C01850=1115.478,64.441,-55.172,179.980,7.501,149.417
C01851=1115.474,64.655,-55.187,179.981,7.504,149.417
C01852=1115.470,64.869,-55.202,179.982,7.508,149.417
C01853=1115.464,65.119,-55.219,179.983,7.512,149.418
C01854=1115.460,65.367,-55.236,179.984,7.516,149.418
C01855=1115.454,65.617,-55.254,179.985,7.520,149.419
C01856=1115.450,65.867,-55.270,179.987,7.524,149.420
C01857=1115.445,66.116,-55.288,179.988,7.528,149.420
C01858=1115.440,66.366,-55.306,179.990,7.532,149.421
C01859=1115.436,66.615,-55.323,179.991,7.536,149.421
C01860=1115.430,66.864,-55.340,179.993,7.540,149.421
C01861=1115.425,67.114,-55.358,179.993,7.543,149.422
C01862=1115.421,67.363,-55.375,179.995,7.547,149.423
C01863=1115.415,67.612,-55.392,179.996,7.551,149.423
C01864=1115.410,67.861,-55.410,179.997,7.556,149.424
C01865=1115.406,68.111,-55.426,179.999,7.560,149.424
C01866=1115.401,68.360,-55.444,-179.999,7.563,149.425
C01867=1115.396,68.610,-55.462,-179.998,7.568,149.425
C01868=1115.391,68.859,-55.479,-179.997,7.572,149.426
C01869=1115.386,69.108,-55.496,-179.995,7.575,149.426
C01870=1115.381,69.358,-55.514,-179.994,7.580,149.427
C01871=1115.376,69.607,-55.532,-179.993,7.583,149.427
C01872=1115.372,69.856,-55.549,-179.991,7.587,149.428
C01873=1115.367,70.106,-55.566,-179.990,7.591,149.428
C01874=1115.362,70.355,-55.584,-179.989,7.595,149.429
C01875=1115.357,70.604,-55.602,-179.987,7.599,149.429
C01876=1115.352,70.854,-55.619,-179.986,7.603,149.430
C01877=1115.347,71.103,-55.637,-179.985,7.607,149.430
C01878=1115.342,71.353,-55.654,-179.983,7.611,149.431
C01879=1115.337,71.602,-55.672,-179.981,7.615,149.431
C01880=1115.333,71.851,-55.689,-179.980,7.619,149.432
C01881=1115.328,72.101,-55.707,-179.979,7.623,149.432
C01882=1115.323,72.350,-55.725,-179.977,7.627,149.433
C01883=1115.318,72.599,-55.743,-179.977,7.630,149.433
C01884=1115.313,72.849,-55.760,-179.975,7.634,149.434
C01885=1115.308,73.098,-55.778,-179.973,7.638,149.434
C01886=1115.304,73.347,-55.795,-179.972,7.643,149.435
C01887=1115.299,73.597,-55.813,-179.971,7.646,149.435
C01888=1115.294,73.846,-55.831,-179.969,7.650,149.436
C01889=1115.289,74.095,-55.848,-179.968,7.654,149.436
C01890=1115.284,74.344,-55.866,-179.967,7.659,149.437
C01891=1115.279,74.594,-55.884,-179.965,7.662,149.437
C01892=1115.274,74.843,-55.902,-179.963,7.666,149.437
C01893=1115.270,75.092,-55.919,-179.962,7.670,149.438
C01894=1115.265,75.341,-55.937,-179.961,7.675,149.439
C01895=1115.259,75.591,-55.954,-179.959,7.678,149.439
C01896=1115.254,75.840,-55.972,-179.958,7.682,149.439
C01897=1115.250,76.089,-55.990,-179.956,7.686,149.440
C01898=1115.245,76.338,-56.008,-179.955,7.690,149.440
C01899=1115.240,76.588,-56.026,-179.954,7.694,149.441
C01900=1115.235,76.837,-56.044,-179.952,7.698,149.441
C01901=1115.231,77.052,-56.060,-179.951,7.701,149.442
C01902=1115.227,77.266,-56.075,-179.951,7.704,149.442
C01903=1115.222,77.480,-56.090,-179.950,7.707,149.443
C01904=1115.219,77.694,-56.106,-179.949,7.710,149.443
C01905=1115.214,77.908,-56.121,-179.948,7.714,149.444
C01906=1115.210,78.123,-56.136,-179.947,7.717,149.444
C01907=1115.206,78.337,-56.152,-179.946,7.720,149.445
C01908=1115.201,78.551,-56.167,-179.946,7.723,149.445
C01909=1115.196,78.800,-56.185,-179.944,7.728,149.446
C01910=1115.192,79.049,-56.203,-179.943,7.731,149.446
C01911=1115.187,79.298,-56.221,-179.942,7.735,149.447
C01912=1115.182,79.548,-56.239,-179.941,7.738,149.447
C01913=1115.177,79.798,-56.257,-179.940,7.742,149.448
C01914=1115.173,80.047,-56.275,-179.939,7.745,149.448
C01915=1115.168,80.296,-56.293,-179.938,7.750,149.449
C01916=1115.163,80.545,-56.311,-179.937,7.753,149.450
C01917=1115.158,80.794,-56.329,-179.936,7.757,149.450
C01918=1115.153,81.043,-56.347,-179.935,7.760,149.451
C01919=1115.149,81.293,-56.366,-179.934,7.764,149.451
C01920=1115.144,81.542,-56.384,-179.933,7.768,149.452
C01921=1115.139,81.792,-56.402,-179.932,7.772,149.452
C01922=1115.133,82.041,-56.420,-179.930,7.776,149.453
C01923=1115.128,82.290,-56.438,-179.930,7.779,149.453
C01924=1115.124,82.540,-56.456,-179.928,7.783,149.454
C01925=1115.119,82.789,-56.474,-179.928,7.787,149.455
C01926=1115.114,83.039,-56.492,-179.926,7.791,149.455
C01927=1115.109,83.288,-56.510,-179.925,7.795,149.456
C01928=1115.104,83.537,-56.528,-179.924,7.798,149.456
C01929=1115.100,83.786,-56.547,-179.923,7.802,149.457
C01930=1115.095,84.035,-56.565,-179.922,7.805,149.457
C01931=1115.090,84.285,-56.584,-179.920,7.809,149.458
C01932=1115.085,84.534,-56.602,-179.919,7.814,149.458
C01933=1115.080,84.783,-56.620,-179.918,7.817,149.459
C01934=1115.076,85.033,-56.638,-179.917,7.821,149.459
C01935=1115.071,85.282,-56.656,-179.915,7.825,149.460
C01936=1115.066,85.531,-56.675,-179.914,7.828,149.460
C01937=1115.060,85.780,-56.694,-179.913,7.832,149.461
C01938=1115.056,86.030,-56.712,-179.912,7.836,149.461
C01939=1115.051,86.279,-56.730,-179.911,7.840,149.462
C01940=1115.046,86.528,-56.748,-179.910,7.843,149.462
C01941=1115.042,86.777,-56.767,-179.908,7.847,149.463
C01942=1115.037,87.027,-56.785,-179.907,7.852,149.463
C01943=1115.032,87.276,-56.803,-179.906,7.855,149.464
C01944=1115.027,87.526,-56.821,-179.904,7.859,149.464
C01945=1115.022,87.774,-56.840,-179.903,7.863,149.465
C01946=1115.017,88.024,-56.859,-179.902,7.867,149.465
C01947=1115.012,88.273,-56.877,-179.901,7.870,149.466
C01948=1115.008,88.522,-56.896,-179.900,7.874,149.466
C01949=1115.003,88.772,-56.914,-179.898,7.878,149.467
C01950=1114.998,89.021,-56.933,-179.896,7.882,149.467
C01951=1114.993,89.270,-56.951,-179.895,7.885,149.468
C01952=1114.988,89.519,-56.969,-179.894,7.889,149.468
C01953=1114.984,89.769,-56.988,-179.893,7.893,149.469
C01954=1114.978,90.018,-57.007,-179.891,7.897,149.469
C01955=1114.974,90.267,-57.025,-179.889,7.901,149.470
C01956=1114.969,90.517,-57.043,-179.889,7.905,149.470
C01957=1114.964,90.731,-57.060,-179.887,7.908,149.470
C01958=1114.960,90.945,-57.076,-179.886,7.911,149.471
C01959=1114.956,91.159,-57.092,-179.885,7.914,149.471
C01960=1114.953,91.373,-57.108,-179.884,7.917,149.472
C01961=1114.948,91.588,-57.123,-179.882,7.921,149.472
C01962=1114.944,91.801,-57.139,-179.881,7.924,149.473
C01963=1114.939,92.015,-57.156,-179.880,7.927,149.473
C01964=1114.936,92.230,-57.172,-179.879,7.931,149.473
C01965=1114.931,92.479,-57.190,-179.878,7.934,149.474
C01966=1114.926,92.728,-57.209,-179.876,7.938,149.474
C01967=1114.921,92.977,-57.227,-179.875,7.942,149.475
C01968=1114.916,93.226,-57.246,-179.873,7.946,149.475
C01969=1114.911,93.476,-57.265,-179.872,7.950,149.476
C01970=1114.907,93.725,-57.284,-179.870,7.954,149.476
C01971=1114.902,93.974,-57.303,-179.868,7.958,149.477
C01972=1114.897,94.224,-57.321,-179.867,7.962,149.477
C01973=1114.892,94.472,-57.341,-179.866,7.966,149.478
C01974=1114.888,94.722,-57.359,-179.865,7.969,149.478
C01975=1114.883,94.971,-57.378,-179.863,7.973,149.478
C01976=1114.878,95.221,-57.397,-179.861,7.977,149.479
C01977=1114.873,95.470,-57.415,-179.860,7.981,149.479
C01978=1114.868,95.718,-57.435,-179.858,7.985,149.480
C01979=1114.864,95.968,-57.453,-179.857,7.989,149.480
C01980=1114.858,96.217,-57.472,-179.855,7.992,149.481
C01981=1114.854,96.466,-57.491,-179.853,7.996,149.481
C01982=1114.849,96.716,-57.510,-179.852,8.000,149.482
C01983=1114.845,96.965,-57.529,-179.850,8.004,149.482
C01984=1114.839,97.214,-57.548,-179.848,8.008,149.482
C01985=1114.835,97.464,-57.567,-179.847,8.011,149.483
C01986=1114.830,97.713,-57.586,-179.845,8.015,149.483
C01987=1114.826,97.962,-57.605,-179.843,8.019,149.483
C01988=1114.820,98.212,-57.624,-179.842,8.023,149.484
C01989=1114.815,98.460,-57.643,-179.840,8.027,149.484
C01990=1114.811,98.710,-57.662,-179.839,8.031,149.485
C01991=1114.805,98.959,-57.681,-179.837,8.035,149.485
C01992=1114.801,99.208,-57.700,-179.835,8.038,149.485
C01993=1114.796,99.457,-57.719,-179.833,8.042,149.486
C01994=1114.792,99.707,-57.738,-179.832,8.046,149.486
C01995=1114.787,99.956,-57.758,-179.830,8.050,149.487
C01996=1114.782,100.205,-57.777,-179.828,8.054,149.487
C01997=1114.777,100.455,-57.795,-179.826,8.057,149.487
C01998=1114.772,100.704,-57.814,-179.825,8.061,149.488
C01999=1114.767,100.953,-57.834,-179.823,8.065,149.488
C02000=1114.763,101.202,-57.853,-179.822,8.069,149.489
C02001=1114.758,101.451,-57.872,-179.820,8.073,149.489
C02002=1114.753,101.700,-57.891,-179.818,8.076,149.489
C02003=1114.748,101.950,-57.911,-179.816,8.080,149.490
C02004=1114.743,102.198,-57.930,-179.814,8.084,149.490
C02005=1114.738,102.448,-57.950,-179.813,8.088,149.490
C02006=1114.734,102.697,-57.968,-179.811,8.092,149.491
C02007=1114.729,102.947,-57.987,-179.809,8.095,149.491
C02008=1114.724,103.196,-58.007,-179.807,8.099,149.492
C02009=1114.719,103.445,-58.026,-179.806,8.103,149.492
C02010=1114.715,103.694,-58.045,-179.804,8.106,149.492
C02011=1114.709,103.943,-58.065,-179.802,8.110,149.493
C02012=1114.704,104.193,-58.084,-179.800,8.114,149.493
C02013=1114.701,104.406,-58.101,-179.798,8.118,149.493
C02014=1114.696,104.621,-58.118,-179.796,8.121,149.493
C02015=1114.693,104.834,-58.135,-179.795,8.124,149.494
C02016=1114.688,105.049,-58.151,-179.793,8.127,149.494
C02017=1114.685,105.263,-58.167,-179.792,8.130,149.494
C02018=1114.680,105.476,-58.185,-179.790,8.134,149.495
C02019=1114.676,105.691,-58.201,-179.788,8.137,149.495
C02020=1114.672,105.904,-58.218,-179.787,8.141,149.495
C02021=1114.667,106.154,-58.238,-179.785,8.144,149.495
C02022=1114.663,106.403,-58.257,-179.783,8.148,149.496
C02023=1114.658,106.652,-58.276,-179.781,8.151,149.496
C02024=1114.653,106.901,-58.296,-179.779,8.155,149.496
C02025=1114.648,107.151,-58.315,-179.777,8.159,149.497
C02026=1114.643,107.400,-58.335,-179.775,8.162,149.497
C02027=1114.639,107.649,-58.355,-179.773,8.167,149.497
C02028=1114.634,107.898,-58.374,-179.771,8.171,149.498
C02029=1114.629,108.147,-58.394,-179.769,8.174,149.498
C02030=1114.625,108.397,-58.413,-179.767,8.178,149.498
C02031=1114.619,108.646,-58.433,-179.765,8.181,149.498
C02032=1114.615,108.895,-58.453,-179.763,8.185,149.499
C02033=1114.610,109.144,-58.473,-179.761,8.189,149.499
C02034=1114.605,109.393,-58.492,-179.759,8.193,149.499
C02035=1114.600,109.643,-58.512,-179.757,8.196,149.499
C02036=1114.596,109.891,-58.532,-179.754,8.200,149.500
C02037=1114.591,110.141,-58.552,-179.753,8.204,149.500
C02038=1114.586,110.390,-58.571,-179.751,8.207,149.500
C02039=1114.581,110.639,-58.591,-179.748,8.211,149.501
C02040=1114.576,110.888,-58.611,-179.746,8.215,149.501
C02041=1114.572,111.138,-58.630,-179.744,8.218,149.501
C02042=1114.567,111.386,-58.650,-179.742,8.222,149.501
C02043=1114.563,111.636,-58.670,-179.741,8.225,149.502
C02044=1114.558,111.885,-58.689,-179.739,8.228,149.502
C02045=1114.553,112.134,-58.710,-179.737,8.232,149.502
C02046=1114.547,112.383,-58.730,-179.735,8.236,149.503
C02047=1114.543,112.632,-58.750,-179.733,8.239,149.503
C02048=1114.538,112.882,-58.770,-179.732,8.242,149.503
C02049=1114.534,113.131,-58.790,-179.730,8.246,149.503
C02050=1114.529,113.380,-58.810,-179.728,8.249,149.504
C02051=1114.524,113.628,-58.830,-179.726,8.253,149.504
C02052=1114.519,113.878,-58.849,-179.724,8.257,149.504
C02053=1114.515,114.128,-58.869,-179.723,8.260,149.505
C02054=1114.510,114.377,-58.889,-179.721,8.263,149.505
C02055=1114.505,114.626,-58.909,-179.719,8.267,149.505
C02056=1114.500,114.874,-58.929,-179.717,8.270,149.505
C02057=1114.496,115.123,-58.949,-179.715,8.274,149.506
C02058=1114.491,115.373,-58.969,-179.714,8.277,149.506
C02059=1114.487,115.622,-58.989,-179.712,8.281,149.506
C02060=1114.481,115.872,-59.010,-179.710,8.284,149.507
C02061=1114.477,116.121,-59.030,-179.708,8.288,149.507
C02062=1114.472,116.370,-59.050,-179.707,8.291,149.507
C02063=1114.467,116.619,-59.070,-179.705,8.294,149.507
C02064=1114.463,116.867,-59.090,-179.703,8.298,149.508
C02065=1114.458,117.117,-59.110,-179.701,8.301,149.508
C02066=1114.453,117.366,-59.130,-179.700,8.304,149.508
C02067=1114.448,117.615,-59.151,-179.698,8.308,149.509
C02068=1114.443,117.865,-59.171,-179.696,8.311,149.509
C02069=1114.439,118.079,-59.188,-179.694,8.314,149.509
C02070=1114.435,118.292,-59.206,-179.693,8.317,149.509
C02071=1114.431,118.506,-59.222,-179.691,8.319,149.509
C02072=1114.427,118.720,-59.240,-179.690,8.323,149.510
C02073=1114.424,118.934,-59.258,-179.688,8.326,149.510
C02074=1114.419,119.148,-59.275,-179.687,8.329,149.510
C02075=1114.415,119.362,-59.292,-179.685,8.331,149.511
C02076=1114.411,119.575,-59.310,-179.684,8.334,149.511
C02077=1114.406,119.824,-59.330,-179.682,8.338,149.511
C02078=1114.402,120.074,-59.350,-179.680,8.341,149.511
C02079=1114.396,120.323,-59.371,-179.678,8.345,149.512
C02080=1114.392,120.572,-59.391,-179.677,8.348,149.512
C02081=1114.388,120.821,-59.412,-179.675,8.351,149.512
C02082=1114.383,121.070,-59.432,-179.673,8.355,149.512
C02083=1114.378,121.320,-59.452,-179.671,8.359,149.513
C02084=1114.373,121.569,-59.473,-179.670,8.361,149.513
C02085=1114.369,121.818,-59.493,-179.668,8.365,149.513
C02086=1114.364,122.067,-59.514,-179.666,8.368,149.513
C02087=1114.359,122.316,-59.534,-179.664,8.371,149.514
C02088=1114.355,122.565,-59.555,-179.662,8.375,149.514
C02089=1114.350,122.814,-59.576,-179.660,8.378,149.514
C02090=1114.345,123.064,-59.595,-179.659,8.381,149.515
C02091=1114.340,123.313,-59.616,-179.657,8.385,149.515
C02092=1114.335,123.562,-59.637,-179.655,8.388,149.515
C02093=1114.331,123.811,-59.657,-179.653,8.392,149.515
C02094=1114.326,124.060,-59.677,-179.652,8.395,149.516
C02095=1114.321,124.309,-59.698,-179.650,8.398,149.516
C02096=1114.317,124.558,-59.719,-179.648,8.402,149.516
C02097=1114.312,124.807,-59.739,-179.647,8.405,149.517
C02098=1114.307,125.056,-59.760,-179.645,8.408,149.517
C02099=1114.303,125.305,-59.780,-179.642,8.412,149.517
C02100=1114.297,125.555,-59.801,-179.642,8.415,149.517
C02101=1114.293,125.804,-59.822,-179.639,8.418,149.518
C02102=1114.289,126.053,-59.842,-179.637,8.422,149.518
C02103=1114.283,126.302,-59.863,-179.636,8.425,149.518
C02104=1114.279,126.551,-59.883,-179.634,8.428,149.518
C02105=1114.274,126.800,-59.904,-179.632,8.432,149.519
C02106=1114.269,127.049,-59.925,-179.631,8.435,149.519
C02107=1114.264,127.298,-59.946,-179.629,8.438,149.519
C02108=1114.260,127.547,-59.966,-179.627,8.442,149.519
C02109=1114.255,127.797,-59.987,-179.625,8.446,149.520
C02110=1114.251,128.045,-60.009,-179.624,8.448,149.520
C02111=1114.246,128.295,-60.030,-179.622,8.452,149.520
C02112=1114.241,128.544,-60.050,-179.619,8.455,149.521
C02113=1114.236,128.793,-60.071,-179.618,8.458,149.521
C02114=1114.232,129.042,-60.091,-179.616,8.462,149.521
C02115=1114.227,129.291,-60.112,-179.614,8.465,149.521
C02116=1114.222,129.540,-60.133,-179.613,8.468,149.522
C02117=1114.217,129.789,-60.154,-179.611,8.472,149.522
C02118=1114.213,130.038,-60.175,-179.609,8.475,149.522
C02119=1114.208,130.288,-60.196,-179.608,8.478,149.523
C02120=1114.204,130.537,-60.216,-179.606,8.482,149.523
C02121=1114.199,130.785,-60.238,-179.604,8.485,149.523
C02122=1114.194,131.034,-60.259,-179.603,8.488,149.524
C02123=1114.189,131.283,-60.279,-179.601,8.492,149.524
C02124=1114.184,131.533,-60.300,-179.599,8.496,149.524
C02125=1114.181,131.747,-60.319,-179.597,8.498,149.524
C02126=1114.177,131.960,-60.336,-179.596,8.501,149.525
C02127=1114.173,132.173,-60.354,-179.595,8.504,149.525
C02128=1114.168,132.388,-60.373,-179.593,8.506,149.525
C02129=1114.164,132.601,-60.391,-179.592,8.509,149.525
C02130=1114.160,132.815,-60.408,-179.590,8.512,149.526
C02131=1114.157,133.029,-60.427,-179.589,8.515,149.526
C02132=1114.152,133.243,-60.445,-179.587,8.518,149.526
C02133=1114.148,133.492,-60.466,-179.586,8.521,149.526
C02134=1114.143,133.742,-60.487,-179.584,8.525,149.527
C02135=1114.138,133.991,-60.508,-179.582,8.528,149.527
C02136=1114.134,134.239,-60.529,-179.581,8.531,149.527
C02137=1114.129,134.488,-60.550,-179.579,8.535,149.528
C02138=1114.124,134.737,-60.572,-179.576,8.538,149.528
C02139=1114.120,134.987,-60.593,-179.575,8.541,149.528
C02140=1114.115,135.236,-60.614,-179.573,8.545,149.528
C02141=1114.110,135.485,-60.635,-179.571,8.548,149.529
C02142=1114.105,135.733,-60.656,-179.570,8.551,149.529
C02143=1114.101,135.983,-60.678,-179.568,8.555,149.529
C02144=1114.096,136.232,-60.699,-179.567,8.558,149.530
C02145=1114.091,136.481,-60.720,-179.565,8.561,149.530
C02146=1114.087,136.730,-60.741,-179.563,8.565,149.530
C02147=1114.082,136.979,-60.763,-179.562,8.568,149.530
C02148=1114.077,137.228,-60.784,-179.560,8.572,149.531
C02149=1114.072,137.477,-60.805,-179.558,8.575,149.531
C02150=1114.068,137.726,-60.826,-179.556,8.578,149.531
C02151=1114.064,137.975,-60.848,-179.555,8.582,149.532
C02152=1114.058,138.224,-60.869,-179.553,8.585,149.532
C02153=1114.054,138.473,-60.890,-179.551,8.588,149.532
C02154=1114.050,138.722,-60.912,-179.550,8.592,149.533
C02155=1114.045,138.971,-60.933,-179.548,8.595,149.533
C02156=1114.040,139.220,-60.955,-179.547,8.598,149.533
C02157=1114.035,139.469,-60.976,-179.545,8.602,149.534
C02158=1114.031,139.719,-60.998,-179.542,8.605,149.534
C02159=1114.026,139.967,-61.019,-179.541,8.608,149.534
C02160=1114.021,140.216,-61.040,-179.539,8.612,149.535
C02161=1114.017,140.466,-61.062,-179.538,8.616,149.535
C02162=1114.012,140.714,-61.083,-179.536,8.618,149.535
C02163=1114.007,140.963,-61.104,-179.535,8.622,149.536
C02164=1114.003,141.213,-61.126,-179.533,8.625,149.536
C02165=1113.998,141.461,-61.148,-179.531,8.629,149.536
C02166=1113.993,141.711,-61.169,-179.529,8.632,149.537
C02167=1113.989,141.960,-61.190,-179.528,8.635,149.537
C02168=1113.984,142.208,-61.212,-179.526,8.639,149.537
C02169=1113.980,142.458,-61.234,-179.524,8.642,149.537
C02170=1113.975,142.707,-61.255,-179.523,8.646,149.538
C02171=1113.970,142.956,-61.277,-179.521,8.649,149.538
C02172=1113.966,143.205,-61.299,-179.520,8.653,149.539
C02173=1113.961,143.454,-61.321,-179.518,8.656,149.539
C02174=1113.956,143.702,-61.342,-179.516,8.659,149.539
C02175=1113.951,143.952,-61.364,-179.514,8.663,149.539
C02176=1113.946,144.201,-61.385,-179.513,8.666,149.540
C02177=1113.942,144.450,-61.407,-179.511,8.670,149.540
C02178=1113.937,144.699,-61.429,-179.510,8.673,149.541
C02179=1113.932,144.947,-61.451,-179.508,8.676,149.541
C02180=1113.928,145.197,-61.473,-179.507,8.680,149.541
C02181=1113.924,145.410,-61.491,-179.505,8.683,149.541
C02182=1113.920,145.624,-61.510,-179.503,8.686,149.542
C02183=1113.917,145.838,-61.528,-179.501,8.690,149.542
C02184=1113.912,146.051,-61.547,-179.500,8.692,149.542
C02185=1113.909,146.265,-61.566,-179.497,8.696,149.542
C02186=1113.904,146.479,-61.584,-179.495,8.699,149.543
C02187=1113.901,146.693,-61.603,-179.494,8.702,149.543
C02188=1113.896,146.906,-61.622,-179.492,8.706,149.543
C02189=1113.892,147.156,-61.644,-179.490,8.709,149.543
C02190=1113.887,147.404,-61.665,-179.488,8.713,149.544
C02191=1113.883,147.654,-61.687,-179.486,8.716,149.544
C02192=1113.878,147.902,-61.709,-179.484,8.720,149.544
C02193=1113.874,148.152,-61.731,-179.481,8.723,149.544
C02194=1113.868,148.400,-61.753,-179.479,8.727,149.544
C02195=1113.864,148.650,-61.775,-179.477,8.731,149.545
C02196=1113.859,148.898,-61.797,-179.475,8.734,149.545
C02197=1113.855,149.148,-61.819,-179.473,8.738,149.545
C02198=1113.850,149.396,-61.841,-179.470,8.741,149.545
C02199=1113.845,149.646,-61.863,-179.468,8.745,149.546
C02200=1113.841,149.894,-61.885,-179.466,8.748,149.546
C02201=1113.836,150.144,-61.907,-179.464,8.752,149.546
C02202=1113.831,150.392,-61.930,-179.462,8.755,149.546
C02203=1113.827,150.641,-61.952,-179.460,8.758,149.546
C02204=1113.822,150.890,-61.973,-179.457,8.763,149.547
C02205=1113.818,151.139,-61.995,-179.455,8.766,149.547
C02206=1113.813,151.388,-62.017,-179.453,8.770,149.547
C02207=1113.808,151.638,-62.040,-179.451,8.773,149.547
C02208=1113.803,151.886,-62.062,-179.449,8.776,149.548
C02209=1113.799,152.135,-62.084,-179.446,8.780,149.548
C02210=1113.794,152.384,-62.106,-179.444,8.783,149.548
C02211=1113.789,152.633,-62.128,-179.442,8.787,149.548
C02212=1113.785,152.883,-62.151,-179.440,8.790,149.548
C02213=1113.780,153.131,-62.173,-179.438,8.794,149.549
C02214=1113.776,153.380,-62.195,-179.435,8.797,149.549
C02215=1113.770,153.629,-62.217,-179.433,8.800,149.549
C02216=1113.766,153.878,-62.240,-179.431,8.804,149.549
C02217=1113.762,154.127,-62.262,-179.429,8.807,149.549
C02218=1113.756,154.376,-62.284,-179.426,8.810,149.549
C02219=1113.752,154.625,-62.307,-179.424,8.814,149.550
C02220=1113.748,154.873,-62.329,-179.422,8.817,149.550
C02221=1113.743,155.123,-62.351,-179.420,8.821,149.550
C02222=1113.739,155.372,-62.374,-179.418,8.824,149.550
C02223=1113.734,155.620,-62.396,-179.416,8.827,149.550
C02224=1113.729,155.870,-62.419,-179.413,8.831,149.551
C02225=1113.725,156.119,-62.441,-179.412,8.833,149.551
C02226=1113.720,156.367,-62.463,-179.410,8.837,149.551
C02227=1113.715,156.616,-62.486,-179.407,8.840,149.551
C02228=1113.711,156.866,-62.508,-179.405,8.843,149.551
C02229=1113.706,157.114,-62.531,-179.403,8.847,149.551
C02230=1113.701,157.363,-62.553,-179.400,8.850,149.551
C02231=1113.697,157.612,-62.576,-179.398,8.853,149.552
C02232=1113.692,157.861,-62.598,-179.396,8.857,149.552
C02233=1113.688,158.110,-62.621,-179.394,8.860,149.552
C02234=1113.684,158.359,-62.643,-179.392,8.863,149.552
C02235=1113.678,158.607,-62.666,-179.389,8.866,149.552
C02236=1113.674,158.857,-62.688,-179.387,8.870,149.552
C02237=1113.670,159.070,-62.708,-179.385,8.872,149.552
C02238=1113.666,159.285,-62.727,-179.384,8.875,149.553
C02239=1113.662,159.497,-62.747,-179.382,8.877,149.553
C02240=1113.658,159.711,-62.766,-179.380,8.881,149.553
C02241=1113.654,159.925,-62.786,-179.378,8.883,149.553
C02242=1113.650,160.139,-62.805,-179.376,8.886,149.553
C02243=1113.646,160.352,-62.825,-179.374,8.889,149.553
C02244=1113.642,160.566,-62.844,-179.372,8.892,149.553
C02245=1113.638,160.814,-62.867,-179.370,8.895,149.553
C02246=1113.633,161.064,-62.890,-179.368,8.898,149.554
C02247=1113.629,161.313,-62.912,-179.365,8.901,149.554
C02248=1113.623,161.561,-62.935,-179.364,8.904,149.554
C02249=1113.620,161.810,-62.958,-179.361,8.907,149.554
C02250=1113.614,162.060,-62.980,-179.359,8.911,149.554
C02251=1113.611,162.308,-63.003,-179.357,8.914,149.554
C02252=1113.606,162.557,-63.027,-179.354,8.917,149.554
C02253=1113.601,162.806,-63.050,-179.352,8.920,149.555
C02254=1113.596,163.055,-63.072,-179.350,8.923,149.555
C02255=1113.592,163.304,-63.095,-179.348,8.926,149.555
C02256=1113.588,163.553,-63.118,-179.345,8.929,149.555
C02257=1113.583,163.802,-63.141,-179.343,8.933,149.555
C02258=1113.578,164.050,-63.163,-179.341,8.936,149.555
C02259=1113.573,164.299,-63.186,-179.339,8.938,149.555
C02260=1113.569,164.548,-63.209,-179.337,8.942,149.555
C02261=1113.565,164.797,-63.232,-179.334,8.945,149.555
C02262=1113.560,165.046,-63.256,-179.332,8.948,149.556
C02263=1113.555,165.295,-63.279,-179.330,8.951,149.556
C02264=1113.551,165.543,-63.301,-179.328,8.954,149.556
C02265=1113.546,165.793,-63.324,-179.326,8.957,149.556
C02266=1113.541,166.042,-63.347,-179.323,8.960,149.556
C02267=1113.537,166.291,-63.370,-179.321,8.964,149.556
C02268=1113.532,166.540,-63.393,-179.319,8.966,149.556
C02269=1113.528,166.789,-63.417,-179.317,8.969,149.556
C02270=1113.523,167.037,-63.439,-179.315,8.973,149.557
C02271=1113.518,167.286,-63.463,-179.312,8.976,149.557
C02272=1113.514,167.535,-63.486,-179.311,8.979,149.557
C02273=1113.509,167.784,-63.509,-179.308,8.982,149.557
C02274=1113.505,168.033,-63.532,-179.306,8.985,149.557
C02275=1113.500,168.282,-63.555,-179.304,8.988,149.557
C02276=1113.496,168.531,-63.579,-179.302,8.991,149.557
C02277=1113.491,168.780,-63.602,-179.299,8.994,149.557
C02278=1113.487,169.028,-63.625,-179.297,8.997,149.557
C02279=1113.482,169.277,-63.648,-179.295,9.000,149.558
C02280=1113.477,169.526,-63.671,-179.293,9.003,149.558
C02281=1113.472,169.775,-63.695,-179.291,9.006,149.558
C02282=1113.468,170.024,-63.718,-179.288,9.009,149.558
C02283=1113.463,170.273,-63.741,-179.286,9.012,149.558
C02284=1113.459,170.522,-63.764,-179.284,9.015,149.558
C02285=1113.455,170.770,-63.788,-179.282,9.018,149.558
C02286=1113.450,171.019,-63.812,-179.280,9.021,149.558
C02287=1113.445,171.268,-63.835,-179.278,9.024,149.558
C02288=1113.440,171.517,-63.858,-179.275,9.027,149.558
C02289=1113.436,171.766,-63.882,-179.273,9.030,149.559
C02290=1113.432,172.015,-63.904,-179.271,9.033,149.559
C02291=1113.427,172.263,-63.928,-179.269,9.036,149.559
C02292=1113.423,172.512,-63.952,-179.266,9.039,149.559
C02293=1113.419,172.726,-63.972,-179.264,9.041,149.559
C02294=1113.414,172.940,-63.992,-179.263,9.044,149.559
C02295=1113.411,173.153,-64.012,-179.261,9.047,149.559
C02296=1113.407,173.366,-64.032,-179.259,9.049,149.559
C02297=1113.403,173.580,-64.053,-179.257,9.052,149.559
C02298=1113.399,173.794,-64.073,-179.255,9.055,149.559
C02299=1113.395,174.007,-64.092,-179.253,9.057,149.559
C02300=1113.392,174.220,-64.113,-179.251,9.059,149.559
C02301=1113.387,174.469,-64.136,-179.249,9.063,149.560
C02302=1113.382,174.718,-64.160,-179.247,9.065,149.560
C02303=1113.378,174.967,-64.184,-179.245,9.068,149.560
C02304=1113.373,175.216,-64.207,-179.243,9.072,149.560
C02305=1113.368,175.465,-64.230,-179.241,9.074,149.560
C02306=1113.364,175.713,-64.254,-179.238,9.077,149.560
C02307=1113.359,175.962,-64.278,-179.236,9.081,149.560
C02308=1113.355,176.211,-64.301,-179.234,9.083,149.560
C02309=1113.350,176.460,-64.325,-179.232,9.086,149.560
C02310=1113.345,176.709,-64.349,-179.230,9.089,149.561
C02311=1113.341,176.957,-64.373,-179.228,9.092,149.561
C02312=1113.336,177.206,-64.396,-179.225,9.095,149.561
C02313=1113.332,177.454,-64.420,-179.224,9.098,149.561
C02314=1113.328,177.704,-64.444,-179.221,9.101,149.561
C02315=1113.323,177.953,-64.467,-179.219,9.104,149.561
C02316=1113.319,178.202,-64.491,-179.217,9.106,149.561
C02317=1113.314,178.451,-64.515,-179.215,9.110,149.561
C02318=1113.309,178.699,-64.539,-179.212,9.113,149.561
C02319=1113.304,178.948,-64.563,-179.210,9.115,149.561
C02320=1113.300,179.197,-64.587,-179.208,9.119,149.562
C02321=1113.295,179.446,-64.610,-179.206,9.122,149.562
C02322=1113.291,179.694,-64.634,-179.203,9.125,149.562
C02323=1113.287,179.943,-64.659,-179.201,9.128,149.562
C02324=1113.282,180.192,-64.682,-179.198,9.131,149.562
C02325=1113.278,180.441,-64.706,-179.195,9.134,149.562
C02326=1113.273,180.690,-64.729,-179.193,9.137,149.562
C02327=1113.269,180.938,-64.753,-179.190,9.140,149.562
C02328=1113.264,181.187,-64.778,-179.189,9.143,149.562
C02329=1113.260,181.437,-64.802,-179.186,9.146,149.562
C02330=1113.255,181.685,-64.826,-179.183,9.149,149.562
C02331=1113.250,181.934,-64.849,-179.181,9.152,149.562
C02332=1113.246,182.183,-64.873,-179.178,9.155,149.562
C02333=1113.241,182.431,-64.898,-179.176,9.158,149.562
C02334=1113.237,182.680,-64.922,-179.173,9.161,149.562
C02335=1113.232,182.930,-64.946,-179.171,9.165,149.562
C02336=1113.228,183.178,-64.970,-179.169,9.167,149.562
C02337=1113.224,183.426,-64.994,-179.166,9.170,149.562
C02338=1113.218,183.676,-65.018,-179.164,9.173,149.562
C02339=1113.214,183.924,-65.042,-179.161,9.176,149.563
C02340=1113.210,184.173,-65.066,-179.159,9.179,149.563
C02341=1113.206,184.422,-65.091,-179.157,9.182,149.563
C02342=1113.201,184.670,-65.115,-179.154,9.185,149.563
C02343=1113.196,184.919,-65.139,-179.152,9.188,149.563
C02344=1113.192,185.168,-65.163,-179.149,9.191,149.563
C02345=1113.187,185.417,-65.188,-179.148,9.193,149.563
C02346=1113.183,185.666,-65.212,-179.145,9.196,149.563
C02347=1113.178,185.914,-65.236,-179.142,9.200,149.563
C02348=1113.174,186.163,-65.260,-179.140,9.203,149.563
C02349=1113.170,186.377,-65.281,-179.138,9.205,149.563
C02350=1113.166,186.590,-65.302,-179.136,9.207,149.563
C02351=1113.162,186.803,-65.322,-179.134,9.210,149.563
C02352=1113.158,187.016,-65.343,-179.132,9.212,149.563
C02353=1113.154,187.230,-65.365,-179.131,9.214,149.563
C02354=1113.151,187.443,-65.385,-179.129,9.217,149.563
C02355=1113.146,187.657,-65.406,-179.126,9.220,149.563
C02356=1113.142,187.870,-65.427,-179.124,9.222,149.563
C02357=1113.138,188.120,-65.451,-179.122,9.224,149.563
C02358=1113.133,188.368,-65.476,-179.119,9.227,149.563
C02359=1113.129,188.617,-65.500,-179.117,9.230,149.563
C02360=1113.124,188.865,-65.524,-179.115,9.233,149.563
C02361=1113.120,189.115,-65.549,-179.112,9.236,149.563
C02362=1113.115,189.363,-65.573,-179.111,9.238,149.563
C02363=1113.110,189.612,-65.598,-179.108,9.241,149.563
C02364=1113.107,189.861,-65.622,-179.106,9.243,149.563
C02365=1113.101,190.110,-65.647,-179.104,9.247,149.564
C02366=1113.097,190.358,-65.671,-179.101,9.250,149.564
C02367=1113.093,190.607,-65.696,-179.100,9.252,149.564
C02368=1113.088,190.855,-65.721,-179.097,9.255,149.564
C02369=1113.084,191.104,-65.745,-179.095,9.258,149.564
C02370=1113.079,191.353,-65.770,-179.093,9.261,149.564
C02371=1113.075,191.601,-65.794,-179.091,9.263,149.564
C02372=1113.071,191.851,-65.819,-179.088,9.266,149.564
C02373=1113.066,192.099,-65.843,-179.086,9.269,149.564
C02374=1113.061,192.348,-65.868,-179.084,9.272,149.564
C02375=1113.057,192.597,-65.892,-179.082,9.274,149.564
C02376=1113.052,192.845,-65.918,-179.079,9.277,149.564
C02377=1113.048,193.095,-65.943,-179.078,9.280,149.564
C02378=1113.044,193.343,-65.967,-179.075,9.283,149.564
C02379=1113.038,193.592,-65.992,-179.074,9.285,149.564
C02380=1113.035,193.841,-66.016,-179.071,9.289,149.564
C02381=1113.030,194.089,-66.041,-179.069,9.291,149.565
C02382=1113.026,194.338,-66.066,-179.067,9.294,149.565
C02383=1113.021,194.587,-66.090,-179.065,9.297,149.565
C02384=1113.016,194.835,-66.116,-179.063,9.300,149.565
C02385=1113.012,195.084,-66.140,-179.061,9.302,149.565
C02386=1113.007,195.333,-66.165,-179.059,9.306,149.565
C02387=1113.003,195.582,-66.189,-179.057,9.308,149.565
C02388=1112.998,195.830,-66.215,-179.055,9.310,149.565
C02389=1112.994,196.079,-66.240,-179.053,9.314,149.565
C02390=1112.990,196.328,-66.264,-179.051,9.316,149.566
C02391=1112.985,196.577,-66.290,-179.048,9.319,149.566
C02392=1112.980,196.825,-66.314,-179.045,9.323,149.566
C02393=1112.976,197.074,-66.338,-179.043,9.326,149.566
C02394=1112.972,197.323,-66.364,-179.040,9.329,149.566
C02395=1112.967,197.571,-66.388,-179.037,9.332,149.566
C02396=1112.963,197.820,-66.414,-179.035,9.335,149.566
C02397=1112.958,198.068,-66.439,-179.032,9.338,149.566
C02398=1112.954,198.317,-66.464,-179.029,9.342,149.566
C02399=1112.949,198.566,-66.488,-179.026,9.345,149.566
C02400=1112.945,198.815,-66.513,-179.023,9.348,149.566
C02401=1112.940,199.064,-66.539,-179.021,9.351,149.566
C02402=1112.936,199.312,-66.563,-179.018,9.354,149.566
C02403=1112.932,199.561,-66.589,-179.015,9.357,149.565
C02404=1112.927,199.809,-66.614,-179.013,9.360,149.565
C02405=1112.923,200.023,-66.636,-179.010,9.362,149.565
C02406=1112.919,200.236,-66.657,-179.008,9.365,149.565
C02407=1112.915,200.449,-66.679,-179.005,9.367,149.565
C02408=1112.912,200.663,-66.700,-179.003,9.370,149.565
C02409=1112.908,200.876,-66.722,-179.000,9.373,149.565
C02410=1112.904,201.090,-66.744,-178.998,9.375,149.565
C02411=1112.900,201.302,-66.765,-178.995,9.378,149.565
C02412=1112.896,201.515,-66.787,-178.993,9.380,149.565
C02413=1112.892,201.764,-66.812,-178.990,9.383,149.565
C02414=1112.887,202.014,-66.837,-178.987,9.387,149.565
C02415=1112.883,202.261,-66.862,-178.984,9.389,149.565
C02416=1112.879,202.510,-66.888,-178.981,9.392,149.565
C02417=1112.874,202.759,-66.913,-178.979,9.395,149.565
C02418=1112.870,203.008,-66.938,-178.976,9.398,149.565
C02419=1112.865,203.257,-66.964,-178.973,9.401,149.564
C02420=1112.861,203.505,-66.989,-178.970,9.403,149.564
C02421=1112.856,203.754,-67.015,-178.967,9.407,149.564
C02422=1112.852,204.003,-67.040,-178.964,9.409,149.564
C02423=1112.847,204.251,-67.066,-178.961,9.412,149.564
C02424=1112.844,204.500,-67.091,-178.959,9.415,149.564
C02425=1112.838,204.748,-67.115,-178.956,9.418,149.564
C02426=1112.834,204.997,-67.141,-178.953,9.421,149.564
C02427=1112.830,205.246,-67.167,-178.950,9.423,149.564
C02428=1112.825,205.494,-67.192,-178.947,9.426,149.564
C02429=1112.821,205.743,-67.218,-178.944,9.430,149.564
C02430=1112.817,205.992,-67.244,-178.941,9.433,149.563
C02431=1112.812,206.240,-67.269,-178.938,9.435,149.563
C02432=1112.807,206.489,-67.294,-178.935,9.439,149.563
C02433=1112.803,206.738,-67.320,-178.932,9.441,149.563
C02434=1112.799,206.987,-67.346,-178.930,9.444,149.563
C02435=1112.794,207.235,-67.371,-178.927,9.447,149.563
C02436=1112.790,207.484,-67.397,-178.924,9.450,149.563
C02437=1112.786,207.732,-67.423,-178.921,9.453,149.563
C02438=1112.781,207.981,-67.448,-178.918,9.455,149.563
C02439=1112.776,208.230,-67.474,-178.916,9.458,149.563
C02440=1112.772,208.478,-67.500,-178.913,9.461,149.563
C02441=1112.767,208.727,-67.526,-178.910,9.464,149.563
C02442=1112.763,208.975,-67.551,-178.907,9.468,149.563
C02443=1112.758,209.224,-67.577,-178.904,9.471,149.562
C02444=1112.754,209.473,-67.603,-178.901,9.473,149.562
C02445=1112.750,209.722,-67.629,-178.898,9.476,149.562
C02446=1112.745,209.970,-67.654,-178.895,9.479,149.562
C02447=1112.741,210.219,-67.680,-178.893,9.482,149.562
C02448=1112.736,210.467,-67.707,-178.890,9.485,149.562
C02449=1112.732,210.716,-67.732,-178.887,9.488,149.562
C02450=1112.727,210.964,-67.758,-178.884,9.492,149.562
C02451=1112.723,211.213,-67.784,-178.881,9.495,149.562
C02452=1112.719,211.462,-67.809,-178.878,9.498,149.562
C02453=1112.714,211.711,-67.835,-178.876,9.501,149.562
C02454=1112.710,211.959,-67.862,-178.873,9.503,149.562
C02455=1112.706,212.208,-67.888,-178.870,9.507,149.562
C02456=1112.701,212.456,-67.913,-178.867,9.510,149.562
C02457=1112.696,212.705,-67.939,-178.864,9.513,149.562
C02458=1112.693,212.953,-67.966,-178.862,9.516,149.562
C02459=1112.688,213.202,-67.992,-178.859,9.519,149.562
C02460=1112.683,213.451,-68.018,-178.856,9.523,149.562
C02461=1112.679,213.663,-68.039,-178.854,9.526,149.562
C02462=1112.675,213.877,-68.062,-178.852,9.528,149.562
C02463=1112.672,214.090,-68.084,-178.850,9.530,149.562
C02464=1112.667,214.303,-68.107,-178.848,9.533,149.562
C02465=1112.664,214.516,-68.130,-178.847,9.535,149.563
C02466=1112.661,214.729,-68.152,-178.845,9.538,149.563
C02467=1112.657,214.942,-68.174,-178.843,9.540,149.563
C02468=1112.653,215.156,-68.197,-178.841,9.542,149.563
C02469=1112.648,215.405,-68.223,-178.839,9.545,149.563
C02470=1112.644,215.653,-68.249,-178.837,9.549,149.563
C02471=1112.640,215.902,-68.275,-178.835,9.551,149.563
C02472=1112.635,216.150,-68.302,-178.832,9.554,149.563
C02473=1112.631,216.398,-68.328,-178.830,9.557,149.563
C02474=1112.626,216.647,-68.353,-178.827,9.561,149.564
C02475=1112.622,216.896,-68.380,-178.826,9.563,149.564
C02476=1112.618,217.144,-68.406,-178.823,9.566,149.564
C02477=1112.614,217.393,-68.433,-178.821,9.569,149.564
C02478=1112.609,217.642,-68.459,-178.818,9.573,149.564
C02479=1112.605,217.890,-68.485,-178.817,9.575,149.564
C02480=1112.601,218.139,-68.511,-178.814,9.578,149.564
C02481=1112.596,218.387,-68.538,-178.811,9.581,149.564
C02482=1112.592,218.636,-68.564,-178.809,9.585,149.564
C02483=1112.587,218.885,-68.591,-178.807,9.588,149.564
C02484=1112.583,219.133,-68.618,-178.805,9.590,149.565
C02485=1112.579,219.382,-68.643,-178.802,9.594,149.565
C02486=1112.574,219.630,-68.670,-178.800,9.597,149.565
C02487=1112.570,219.879,-68.696,-178.798,9.600,149.565
C02488=1112.565,220.127,-68.723,-178.795,9.603,149.565
C02489=1112.561,220.376,-68.750,-178.793,9.606,149.565
C02490=1112.556,220.625,-68.776,-178.790,9.609,149.565
C02491=1112.552,220.873,-68.802,-178.788,9.612,149.565
C02492=1112.548,221.122,-68.829,-178.786,9.615,149.565
C02493=1112.544,221.370,-68.855,-178.783,9.618,149.565
C02494=1112.539,221.619,-68.882,-178.781,9.621,149.566
C02495=1112.535,221.867,-68.909,-178.779,9.625,149.566
C02496=1112.530,222.116,-68.935,-178.776,9.628,149.566
C02497=1112.526,222.364,-68.962,-178.774,9.631,149.566
C02498=1112.522,222.613,-68.989,-178.771,9.634,149.566
C02499=1112.517,222.862,-69.015,-178.769,9.637,149.566
C02500=1112.513,223.110,-69.041,-178.766,9.640,149.566
C02501=1112.508,223.358,-69.069,-178.763,9.643,149.566
C02502=1112.504,223.607,-69.095,-178.761,9.646,149.566
C02503=1112.499,223.855,-69.122,-178.758,9.649,149.566
C02504=1112.495,224.104,-69.148,-178.756,9.653,149.566
C02505=1112.491,224.352,-69.175,-178.753,9.656,149.566
C02506=1112.486,224.601,-69.202,-178.751,9.659,149.566
C02507=1112.482,224.849,-69.228,-178.748,9.662,149.566
C02508=1112.477,225.098,-69.255,-178.745,9.665,149.566
C02509=1112.473,225.347,-69.283,-178.743,9.668,149.566
C02510=1112.469,225.595,-69.309,-178.740,9.671,149.566
C02511=1112.464,225.844,-69.336,-178.738,9.674,149.567
C02512=1112.460,226.093,-69.363,-178.735,9.677,149.567
C02513=1112.456,226.341,-69.389,-178.733,9.680,149.567
C02514=1112.451,226.589,-69.416,-178.730,9.683,149.567
C02515=1112.446,226.838,-69.443,-178.727,9.686,149.567
C02516=1112.443,227.086,-69.470,-178.725,9.689,149.567
C02517=1112.439,227.299,-69.493,-178.722,9.692,149.567
C02518=1112.435,227.512,-69.517,-178.720,9.694,149.567
C02519=1112.431,227.726,-69.540,-178.717,9.697,149.567
C02520=1112.428,227.938,-69.563,-178.716,9.700,149.567
C02521=1112.424,228.151,-69.586,-178.713,9.702,149.567
C02522=1112.421,228.364,-69.610,-178.711,9.705,149.567
C02523=1112.416,228.577,-69.632,-178.708,9.708,149.567
C02524=1112.412,228.790,-69.655,-178.706,9.710,149.567
C02525=1112.408,229.039,-69.682,-178.703,9.713,149.567
C02526=1112.404,229.288,-69.709,-178.700,9.716,149.567
C02527=1112.400,229.536,-69.736,-178.697,9.718,149.566
C02528=1112.395,229.785,-69.763,-178.695,9.722,149.566
C02529=1112.391,230.032,-69.791,-178.692,9.724,149.566
C02530=1112.387,230.281,-69.818,-178.689,9.728,149.566
C02531=1112.383,230.530,-69.845,-178.686,9.731,149.566
C02532=1112.378,230.778,-69.872,-178.683,9.734,149.566
C02533=1112.373,231.027,-69.899,-178.680,9.737,149.566
C02534=1112.369,231.275,-69.927,-178.677,9.740,149.566
C02535=1112.364,231.523,-69.954,-178.674,9.742,149.566
C02536=1112.361,231.772,-69.981,-178.672,9.745,149.566
C02537=1112.356,232.021,-70.008,-178.669,9.748,149.566
C02538=1112.352,232.269,-70.036,-178.666,9.751,149.566
C02539=1112.347,232.517,-70.063,-178.664,9.753,149.566
C02540=1112.343,232.766,-70.090,-178.661,9.756,149.566
C02541=1112.339,233.015,-70.117,-178.658,9.759,149.566
C02542=1112.334,233.263,-70.145,-178.655,9.761,149.565
C02543=1112.330,233.511,-70.172,-178.652,9.764,149.565
C02544=1112.326,233.760,-70.200,-178.650,9.767,149.565
C02545=1112.321,234.008,-70.227,-178.647,9.770,149.565
C02546=1112.316,234.257,-70.254,-178.644,9.773,149.565
C02547=1112.312,234.506,-70.282,-178.642,9.775,149.565
C02548=1112.309,234.753,-70.309,-178.639,9.778,149.565
C02549=1112.304,235.002,-70.336,-178.636,9.781,149.565
C02550=1112.300,235.251,-70.364,-178.633,9.783,149.565
C02551=1112.296,235.499,-70.391,-178.630,9.786,149.565
C02552=1112.291,235.747,-70.419,-178.628,9.788,149.565
C02553=1112.287,235.996,-70.447,-178.625,9.791,149.564
C02554=1112.283,236.244,-70.474,-178.622,9.794,149.565
C02555=1112.278,236.493,-70.502,-178.620,9.797,149.564
C02556=1112.274,236.742,-70.529,-178.617,9.799,149.564
C02557=1112.269,236.990,-70.557,-178.614,9.801,149.564
C02558=1112.265,237.238,-70.585,-178.611,9.804,149.564
C02559=1112.261,237.487,-70.612,-178.609,9.807,149.564
C02560=1112.256,237.735,-70.640,-178.606,9.809,149.564
C02561=1112.252,237.983,-70.667,-178.604,9.812,149.564
C02562=1112.248,238.232,-70.695,-178.601,9.814,149.564
C02563=1112.243,238.480,-70.722,-178.598,9.817,149.564
C02564=1112.239,238.728,-70.750,-178.596,9.820,149.564
C02565=1112.235,238.977,-70.778,-178.593,9.822,149.564
C02566=1112.231,239.225,-70.805,-178.591,9.825,149.563
C02567=1112.226,239.474,-70.834,-178.588,9.827,149.563
C02568=1112.221,239.723,-70.861,-178.586,9.830,149.563
C02569=1112.217,239.971,-70.889,-178.583,9.832,149.563
C02570=1112.213,240.219,-70.917,-178.580,9.835,149.563
C02571=1112.209,240.468,-70.944,-178.578,9.838,149.563
C02572=1112.205,240.716,-70.972,-178.575,9.840,149.563
C02573=1112.202,240.929,-70.997,-178.573,9.842,149.563
C02574=1112.197,241.142,-71.021,-178.571,9.845,149.563
C02575=1112.193,241.355,-71.044,-178.568,9.847,149.563
C02576=1112.190,241.567,-71.068,-178.567,9.849,149.563
C02577=1112.186,241.780,-71.092,-178.564,9.851,149.563
C02578=1112.182,241.993,-71.115,-178.562,9.853,149.563
C02579=1112.179,242.206,-71.140,-178.560,9.855,149.563
C02580=1112.175,242.419,-71.164,-178.558,9.858,149.563
C02581=1112.171,242.668,-71.192,-178.555,9.860,149.563
C02582=1112.166,242.916,-71.220,-178.553,9.863,149.563
C02583=1112.163,243.164,-71.248,-178.550,9.865,149.563
C02584=1112.157,243.413,-71.275,-178.548,9.868,149.563
C02585=1112.154,243.662,-71.304,-178.546,9.870,149.563
C02586=1112.149,243.909,-71.331,-178.544,9.873,149.563
C02587=1112.145,244.158,-71.359,-178.541,9.876,149.563
C02588=1112.140,244.406,-71.388,-178.538,9.879,149.563
C02589=1112.137,244.655,-71.416,-178.536,9.881,149.563
C02590=1112.132,244.903,-71.444,-178.533,9.884,149.562
C02591=1112.128,245.152,-71.472,-178.531,9.886,149.563
C02592=1112.123,245.400,-71.500,-178.529,9.889,149.563
C02593=1112.119,245.649,-71.528,-178.527,9.892,149.563
C02594=1112.114,245.897,-71.556,-178.524,9.894,149.563
C02595=1112.111,246.145,-71.584,-178.522,9.897,149.563
C02596=1112.106,246.393,-71.612,-178.520,9.900,149.563
C02597=1112.102,246.642,-71.641,-178.518,9.902,149.563
C02598=1112.097,246.890,-71.668,-178.515,9.905,149.563
C02599=1112.094,247.139,-71.697,-178.513,9.908,149.563
C02600=1112.089,247.387,-71.725,-178.511,9.911,149.563
C02601=1112.085,247.635,-71.753,-178.508,9.913,149.563
C02602=1112.080,247.884,-71.782,-178.504,9.917,149.563
C02603=1112.076,248.132,-71.810,-178.501,9.920,149.563
C02604=1112.072,248.381,-71.838,-178.497,9.924,149.563
C02605=1112.067,248.628,-71.867,-178.493,9.927,149.562
C02606=1112.064,248.877,-71.895,-178.490,9.930,149.562
C02607=1112.059,249.125,-71.923,-178.487,9.933,149.562
C02608=1112.055,249.374,-71.952,-178.483,9.937,149.562
C02609=1112.050,249.622,-71.980,-178.480,9.939,149.562
C02610=1112.046,249.870,-72.008,-178.477,9.942,149.562
C02611=1112.042,250.119,-72.038,-178.473,9.945,149.561
C02612=1112.037,250.366,-72.065,-178.470,9.948,149.561
C02613=1112.033,250.615,-72.094,-178.466,9.950,149.561
C02614=1112.029,250.864,-72.122,-178.464,9.953,149.561
C02615=1112.024,251.112,-72.151,-178.461,9.956,149.561
C02616=1112.021,251.360,-72.179,-178.457,9.958,149.560
C02617=1112.016,251.609,-72.208,-178.454,9.961,149.560
C02618=1112.012,251.857,-72.236,-178.451,9.964,149.560
C02619=1112.008,252.105,-72.265,-178.448,9.966,149.560
C02620=1112.004,252.354,-72.294,-178.446,9.968,149.560
C02621=1111.999,252.602,-72.322,-178.443,9.971,149.560
C02622=1111.995,252.850,-72.351,-178.440,9.974,149.559
C02623=1111.991,253.099,-72.379,-178.437,9.976,149.559
C02624=1111.986,253.347,-72.408,-178.435,9.978,149.559
C02625=1111.982,253.595,-72.437,-178.432,9.980,149.559
C02626=1111.978,253.844,-72.465,-178.430,9.982,149.559
C02627=1111.974,254.092,-72.495,-178.427,9.985,149.559
C02628=1111.969,254.340,-72.523,-178.425,9.987,149.559
C02629=1111.966,254.553,-72.548,-178.422,9.989,149.559
C02630=1111.962,254.766,-72.572,-178.421,9.991,149.559
C02631=1111.958,254.978,-72.597,-178.419,9.993,149.558
C02632=1111.955,255.191,-72.621,-178.417,9.995,149.559
C02633=1111.951,255.404,-72.646,-178.416,9.997,149.559
C02634=1111.948,255.617,-72.671,-178.413,9.999,149.558
C02635=1111.944,255.829,-72.695,-178.412,10.000,149.558
C02636=1111.940,256.043,-72.721,-178.410,10.002,149.559
C02637=1111.936,256.291,-72.748,-178.408,10.006,149.559
C02638=1111.932,256.539,-72.778,-178.405,10.008,149.559
C02639=1111.927,256.788,-72.806,-178.402,10.010,149.558
C02640=1111.924,257.036,-72.835,-178.399,10.013,149.558
C02641=1111.919,257.283,-72.864,-178.397,10.016,149.558
C02642=1111.914,257.532,-72.893,-178.394,10.019,149.558
C02643=1111.911,257.780,-72.922,-178.391,10.022,149.558
C02644=1111.906,258.029,-72.951,-178.388,10.024,149.558
C02645=1111.902,258.277,-72.980,-178.386,10.028,149.558
C02646=1111.897,258.525,-73.009,-178.383,10.030,149.558
C02647=1111.893,258.774,-73.038,-178.380,10.033,149.558
C02648=1111.889,259.022,-73.067,-178.377,10.036,149.558
C02649=1111.885,259.270,-73.096,-178.374,10.038,149.558
C02650=1111.880,259.518,-73.125,-178.371,10.041,149.558
C02651=1111.876,259.766,-73.154,-178.369,10.044,149.558
C02652=1111.873,260.014,-73.183,-178.366,10.046,149.558
C02653=1111.868,260.263,-73.212,-178.363,10.049,149.557
C02654=1111.864,260.512,-73.241,-178.360,10.052,149.557
C02655=1111.860,260.760,-73.271,-178.357,10.055,149.557
C02656=1111.855,261.007,-73.300,-178.354,10.057,149.557
C02657=1111.850,261.256,-73.329,-178.351,10.060,149.557
C02658=1111.846,261.505,-73.358,-178.348,10.063,149.557
C02659=1111.843,261.752,-73.387,-178.345,10.066,149.557
C02660=1111.839,262.001,-73.416,-178.343,10.068,149.557
C02661=1111.834,262.249,-73.446,-178.340,10.071,149.557
C02662=1111.830,262.498,-73.474,-178.337,10.074,149.557
C02663=1111.825,262.745,-73.504,-178.334,10.077,149.556
C02664=1111.821,262.994,-73.533,-178.330,10.079,149.556
C02665=1111.817,263.242,-73.562,-178.327,10.082,149.556
C02666=1111.813,263.490,-73.592,-178.324,10.085,149.556
C02667=1111.808,263.739,-73.621,-178.322,10.087,149.556
C02668=1111.804,263.987,-73.651,-178.319,10.090,149.556
C02669=1111.800,264.235,-73.680,-178.315,10.093,149.555
C02670=1111.796,264.483,-73.710,-178.312,10.095,149.555
C02671=1111.792,264.732,-73.739,-178.309,10.098,149.555
C02672=1111.788,264.980,-73.769,-178.306,10.101,149.555
C02673=1111.782,265.228,-73.797,-178.304,10.103,149.555
C02674=1111.779,265.476,-73.827,-178.301,10.106,149.555
C02675=1111.774,265.724,-73.857,-178.298,10.108,149.555
C02676=1111.770,265.972,-73.886,-178.296,10.110,149.555
C02677=1111.766,266.221,-73.916,-178.293,10.113,149.555
C02678=1111.762,266.469,-73.945,-178.290,10.116,149.554
C02679=1111.758,266.717,-73.974,-178.287,10.118,149.554
C02680=1111.754,266.965,-74.004,-178.284,10.120,149.554
C02681=1111.749,267.214,-74.033,-178.281,10.123,149.554
C02682=1111.745,267.462,-74.063,-178.279,10.126,149.554
C02683=1111.741,267.710,-74.092,-178.276,10.128,149.554
C02684=1111.737,267.958,-74.122,-178.273,10.131,149.554
C02685=1111.733,268.170,-74.147,-178.271,10.132,149.553
C02686=1111.729,268.384,-74.172,-178.268,10.135,149.553
C02687=1111.726,268.596,-74.198,-178.266,10.138,149.553
C02688=1111.722,268.809,-74.224,-178.264,10.140,149.553
C02689=1111.718,269.021,-74.249,-178.262,10.142,149.553
C02690=1111.715,269.234,-74.275,-178.259,10.144,149.553
C02691=1111.711,269.446,-74.300,-178.256,10.146,149.553
C02692=1111.707,269.660,-74.325,-178.254,10.148,149.553
C02693=1111.704,269.907,-74.355,-178.251,10.151,149.553
C02694=1111.699,270.156,-74.385,-178.248,10.154,149.553
C02695=1111.695,270.404,-74.414,-178.245,10.157,149.553
C02696=1111.691,270.652,-74.444,-178.243,10.159,149.552
C02697=1111.686,270.900,-74.475,-178.240,10.161,149.552
C02698=1111.682,271.148,-74.504,-178.237,10.164,149.552
C02699=1111.678,271.397,-74.533,-178.234,10.167,149.552
C02700=1111.674,271.644,-74.564,-178.231,10.170,149.552
C02701=1111.669,271.893,-74.594,-178.229,10.172,149.552
C02702=1111.666,272.142,-74.624,-178.226,10.174,149.552
C02703=1111.662,272.390,-74.654,-178.223,10.177,149.552
C02704=1111.658,272.638,-74.683,-178.220,10.180,149.552
C02705=1111.654,272.885,-74.713,-178.217,10.182,149.551
C02706=1111.649,273.134,-74.743,-178.214,10.185,149.551
C02707=1111.645,273.382,-74.773,-178.211,10.188,149.551
C02708=1111.641,273.630,-74.803,-178.208,10.190,149.551
C02709=1111.636,273.879,-74.833,-178.206,10.193,149.551
C02710=1111.632,274.126,-74.863,-178.203,10.195,149.551
C02711=1111.628,274.375,-74.893,-178.200,10.198,149.551
C02712=1111.624,274.623,-74.923,-178.197,10.201,149.551
C02713=1111.620,274.871,-74.953,-178.194,10.204,149.551
C02714=1111.616,275.119,-74.983,-178.191,10.206,149.550
C02715=1111.612,275.367,-75.013,-178.187,10.209,149.550
C02716=1111.607,275.615,-75.044,-178.185,10.212,149.550
C02717=1111.603,275.864,-75.073,-178.182,10.214,149.550
C02718=1111.599,276.112,-75.104,-178.179,10.216,149.550
C02719=1111.595,276.360,-75.134,-178.176,10.219,149.550
C02720=1111.591,276.608,-75.164,-178.173,10.222,149.550
C02721=1111.586,276.856,-75.195,-178.170,10.224,149.549
C02722=1111.582,277.104,-75.224,-178.167,10.227,149.549
C02723=1111.579,277.353,-75.255,-178.164,10.230,149.549
C02724=1111.574,277.601,-75.285,-178.161,10.233,149.549
C02725=1111.570,277.849,-75.315,-178.158,10.235,149.549
C02726=1111.565,278.097,-75.346,-178.155,10.238,149.549
C02727=1111.561,278.344,-75.376,-178.152,10.240,149.549
C02728=1111.557,278.593,-75.407,-178.150,10.242,149.548
C02729=1111.553,278.841,-75.436,-178.146,10.245,149.548
C02730=1111.548,279.089,-75.467,-178.143,10.248,149.548
C02731=1111.545,279.337,-75.497,-178.141,10.250,149.548
C02732=1111.541,279.586,-75.528,-178.138,10.253,149.548
C02733=1111.536,279.834,-75.558,-178.134,10.256,149.548
C02734=1111.532,280.082,-75.589,-178.131,10.258,149.548
C02735=1111.528,280.330,-75.619,-178.128,10.261,149.547
C02736=1111.524,280.578,-75.650,-178.125,10.263,149.547
C02737=1111.520,280.826,-75.680,-178.122,10.266,149.547
C02738=1111.515,281.074,-75.710,-178.119,10.269,149.547
C02739=1111.511,281.322,-75.740,-178.116,10.271,149.547
C02740=1111.507,281.571,-75.771,-178.112,10.274,149.546
C02741=1111.503,281.783,-75.797,-178.110,10.276,149.546
C02742=1111.500,281.995,-75.824,-178.108,10.278,149.546
C02743=1111.496,282.208,-75.850,-178.105,10.281,149.546
C02744=1111.493,282.420,-75.876,-178.103,10.283,149.546
C02745=1111.490,282.632,-75.902,-178.100,10.284,149.546
C02746=1111.486,282.845,-75.929,-178.097,10.287,149.546
C02747=1111.482,283.058,-75.955,-178.095,10.289,149.545
C02748=1111.479,283.270,-75.981,-178.092,10.291,149.545
C02749=1111.475,283.518,-76.012,-178.089,10.293,149.545
C02750=1111.470,283.766,-76.043,-178.086,10.296,149.545
C02751=1111.466,284.014,-76.073,-178.083,10.299,149.545
C02752=1111.462,284.263,-76.104,-178.080,10.301,149.545
C02753=1111.458,284.511,-76.135,-178.077,10.304,149.545
C02754=1111.454,284.758,-76.165,-178.074,10.306,149.544
C02755=1111.450,285.007,-76.196,-178.071,10.308,149.544
C02756=1111.445,285.255,-76.227,-178.068,10.311,149.544
C02757=1111.441,285.503,-76.258,-178.065,10.314,149.544
C02758=1111.437,285.751,-76.288,-178.062,10.316,149.544
C02759=1111.433,285.999,-76.319,-178.059,10.319,149.543
C02760=1111.429,286.248,-76.350,-178.056,10.322,149.543
C02761=1111.425,286.495,-76.381,-178.052,10.324,149.543
C02762=1111.420,286.743,-76.412,-178.050,10.327,149.543
C02763=1111.416,286.991,-76.443,-178.046,10.329,149.543
C02764=1111.412,287.239,-76.474,-178.044,10.331,149.543
C02765=1111.408,287.488,-76.505,-178.041,10.334,149.542
C02766=1111.404,287.735,-76.536,-178.038,10.336,149.542
C02767=1111.400,287.983,-76.566,-178.035,10.339,149.542
C02768=1111.396,288.232,-76.597,-178.031,10.342,149.542
C02769=1111.391,288.480,-76.628,-178.028,10.344,149.542
C02770=1111.388,288.727,-76.659,-178.025,10.347,149.541
C02771=1111.383,288.975,-76.690,-178.022,10.350,149.541
C02772=1111.379,289.224,-76.721,-178.019,10.351,149.541
C02773=1111.375,289.471,-76.753,-178.016,10.354,149.541
C02774=1111.371,289.720,-76.784,-178.014,10.357,149.541
C02775=1111.367,289.968,-76.815,-178.010,10.359,149.541
C02776=1111.362,290.215,-76.846,-178.007,10.362,149.541
C02777=1111.359,290.464,-76.877,-178.004,10.364,149.540
C02778=1111.354,290.712,-76.908,-178.001,10.367,149.540
C02779=1111.351,290.960,-76.939,-177.998,10.370,149.540
C02780=1111.346,291.208,-76.970,-177.995,10.372,149.540
C02781=1111.342,291.456,-77.002,-177.992,10.374,149.539
C02782=1111.338,291.704,-77.033,-177.989,10.377,149.539
C02783=1111.334,291.952,-77.065,-177.986,10.379,149.539
C02784=1111.329,292.200,-77.095,-177.983,10.382,149.539
C02785=1111.326,292.448,-77.127,-177.980,10.385,149.539
C02786=1111.322,292.696,-77.158,-177.977,10.387,149.539
C02787=1111.317,292.944,-77.190,-177.974,10.390,149.539
C02788=1111.313,293.192,-77.221,-177.970,10.392,149.538
C02789=1111.309,293.440,-77.252,-177.967,10.395,149.538
C02790=1111.306,293.688,-77.283,-177.965,10.397,149.538
C02791=1111.301,293.935,-77.314,-177.962,10.399,149.538
C02792=1111.297,294.184,-77.346,-177.958,10.402,149.538
C02793=1111.293,294.431,-77.377,-177.955,10.405,149.538
C02794=1111.289,294.679,-77.409,-177.953,10.407,149.537
C02795=1111.285,294.928,-77.441,-177.949,10.410,149.537
C02796=1111.280,295.176,-77.472,-177.946,10.413,149.537
C02797=1111.277,295.388,-77.499,-177.944,10.414,149.537
C02798=1111.274,295.600,-77.526,-177.941,10.416,149.537
C02799=1111.270,295.813,-77.553,-177.938,10.419,149.537
C02800=1111.267,296.025,-77.580,-177.936,10.421,149.536
C02801=1111.263,296.237,-77.607,-177.933,10.423,149.536
C02802=1111.260,296.450,-77.634,-177.930,10.425,149.536
C02803=1111.257,296.662,-77.661,-177.928,10.427,149.536
C02804=1111.253,296.875,-77.688,-177.925,10.429,149.536
C02805=1111.249,297.122,-77.719,-177.922,10.432,149.536
C02806=1111.245,297.371,-77.751,-177.919,10.435,149.536
C02807=1111.240,297.619,-77.783,-177.916,10.437,149.535
C02808=1111.236,297.866,-77.814,-177.913,10.440,149.535
C02809=1111.232,298.114,-77.846,-177.910,10.442,149.535
C02810=1111.228,298.362,-77.877,-177.907,10.445,149.535
C02811=1111.224,298.610,-77.909,-177.904,10.447,149.535
C02812=1111.220,298.858,-77.941,-177.901,10.449,149.534
C02813=1111.215,299.106,-77.973,-177.898,10.452,149.534
C02814=1111.212,299.354,-78.005,-177.895,10.455,149.534
C02815=1111.208,299.602,-78.037,-177.892,10.457,149.534
C02816=1111.204,299.849,-78.068,-177.889,10.460,149.534
C02817=1111.200,300.097,-78.100,-177.885,10.462,149.533
C02818=1111.195,300.346,-78.132,-177.883,10.465,149.533
C02819=1111.191,300.594,-78.163,-177.879,10.467,149.533
C02820=1111.187,300.842,-78.195,-177.876,10.470,149.533
C02821=1111.183,301.090,-78.227,-177.873,10.473,149.533
C02822=1111.179,301.338,-78.259,-177.871,10.475,149.533
C02823=1111.175,301.585,-78.291,-177.867,10.477,149.532
C02824=1111.171,301.834,-78.323,-177.864,10.480,149.532
C02825=1111.166,302.082,-78.355,-177.861,10.482,149.532
C02826=1111.162,302.329,-78.386,-177.858,10.485,149.532
C02827=1111.158,302.577,-78.418,-177.855,10.487,149.532
C02828=1111.154,302.825,-78.451,-177.852,10.490,149.532
C02829=1111.151,303.073,-78.483,-177.849,10.493,149.531
C02830=1111.146,303.320,-78.515,-177.846,10.495,149.531
C02831=1111.142,303.569,-78.547,-177.843,10.497,149.531
C02832=1111.138,303.817,-78.579,-177.840,10.500,149.531
C02833=1111.134,304.065,-78.611,-177.837,10.502,149.531
C02834=1111.129,304.312,-78.643,-177.834,10.505,149.531
C02835=1111.126,304.560,-78.675,-177.830,10.508,149.530
C02836=1111.122,304.808,-78.708,-177.827,10.510,149.530
C02837=1111.118,305.056,-78.740,-177.824,10.513,149.530
C02838=1111.113,305.304,-78.771,-177.821,10.515,149.530
C02839=1111.109,305.552,-78.804,-177.818,10.518,149.530
C02840=1111.105,305.800,-78.836,-177.815,10.520,149.529
C02841=1111.101,306.048,-78.869,-177.812,10.522,149.529
C02842=1111.098,306.296,-78.901,-177.809,10.525,149.529
C02843=1111.092,306.543,-78.933,-177.806,10.528,149.529
C02844=1111.089,306.791,-78.965,-177.803,10.530,149.529
C02845=1111.085,307.039,-78.998,-177.800,10.533,149.529
C02846=1111.081,307.287,-79.030,-177.796,10.535,149.528
C02847=1111.077,307.535,-79.061,-177.793,10.538,149.528
C02848=1111.073,307.783,-79.095,-177.790,10.540,149.528
C02849=1111.069,308.031,-79.126,-177.787,10.543,149.528
C02850=1111.065,308.278,-79.159,-177.784,10.545,149.528
C02851=1111.060,308.526,-79.192,-177.782,10.548,149.528
C02852=1111.056,308.774,-79.223,-177.778,10.550,149.527
C02853=1111.053,308.986,-79.251,-177.775,10.553,149.527
C02854=1111.050,309.198,-79.279,-177.773,10.554,149.527
C02855=1111.047,309.411,-79.307,-177.770,10.556,149.527
C02856=1111.043,309.623,-79.335,-177.767,10.559,149.527
C02857=1111.040,309.835,-79.363,-177.765,10.561,149.527
C02858=1111.035,310.048,-79.391,-177.762,10.563,149.526
C02859=1111.032,310.260,-79.418,-177.759,10.566,149.526
C02860=1111.029,310.472,-79.446,-177.757,10.567,149.526
C02861=1111.025,310.720,-79.478,-177.754,10.570,149.526
C02862=1111.021,310.967,-79.511,-177.750,10.573,149.526
C02863=1111.016,311.216,-79.544,-177.748,10.575,149.526
C02864=1111.013,311.463,-79.576,-177.745,10.577,149.525
C02865=1111.009,311.711,-79.609,-177.742,10.580,149.525
C02866=1111.004,311.959,-79.642,-177.739,10.582,149.525
C02867=1111.001,312.207,-79.675,-177.735,10.585,149.525
C02868=1110.997,312.455,-79.707,-177.732,10.587,149.525
C02869=1110.993,312.702,-79.740,-177.729,10.590,149.524
C02870=1110.989,312.950,-79.773,-177.726,10.593,149.524
C02871=1110.985,313.198,-79.805,-177.723,10.595,149.524
C02872=1110.980,313.446,-79.838,-177.720,10.598,149.524
C02873=1110.977,313.694,-79.871,-177.717,10.600,149.524
C02874=1110.973,313.942,-79.903,-177.714,10.602,149.524
C02875=1110.968,314.190,-79.936,-177.711,10.605,149.523
C02876=1110.965,314.437,-79.969,-177.708,10.607,149.523
C02877=1110.961,314.685,-80.001,-177.705,10.610,149.523
C02878=1110.956,314.933,-80.035,-177.701,10.612,149.523
C02879=1110.952,315.181,-80.068,-177.698,10.615,149.523
C02880=1110.949,315.428,-80.100,-177.695,10.618,149.523
C02881=1110.945,315.676,-80.133,-177.692,10.620,149.522
C02882=1110.940,315.924,-80.166,-177.689,10.623,149.522
C02883=1110.936,316.172,-80.199,-177.685,10.625,149.522
C02884=1110.933,316.420,-80.232,-177.683,10.627,149.522
C02885=1110.929,316.667,-80.265,-177.680,10.630,149.522
C02886=1110.925,316.915,-80.298,-177.677,10.632,149.521
C02887=1110.920,317.163,-80.331,-177.674,10.635,149.521
C02888=1110.916,317.410,-80.364,-177.670,10.637,149.521
C02889=1110.913,317.658,-80.396,-177.667,10.640,149.521
C02890=1110.908,317.906,-80.429,-177.664,10.643,149.521
C02891=1110.904,318.154,-80.462,-177.661,10.645,149.521
C02892=1110.900,318.402,-80.496,-177.658,10.648,149.520
C02893=1110.896,318.649,-80.529,-177.654,10.650,149.520
C02894=1110.892,318.898,-80.562,-177.652,10.652,149.520
C02895=1110.888,319.146,-80.595,-177.649,10.655,149.520
C02896=1110.885,319.393,-80.628,-177.646,10.657,149.520
C02897=1110.881,319.641,-80.661,-177.643,10.660,149.520
C02898=1110.877,319.888,-80.694,-177.639,10.662,149.519
C02899=1110.873,320.136,-80.727,-177.636,10.665,149.519
C02900=1110.868,320.384,-80.761,-177.633,10.668,149.519
C02901=1110.865,320.631,-80.794,-177.630,10.670,149.519
C02902=1110.861,320.879,-80.828,-177.627,10.673,149.519
C02903=1110.857,321.127,-80.861,-177.623,10.675,149.518
C02904=1110.853,321.375,-80.894,-177.621,10.677,149.518
C02905=1110.849,321.623,-80.927,-177.618,10.680,149.518
C02906=1110.844,321.870,-80.961,-177.615,10.682,149.518
C02907=1110.840,322.118,-80.994,-177.612,10.685,149.518
C02908=1110.837,322.367,-81.027,-177.608,10.687,149.518
C02909=1110.834,322.578,-81.056,-177.606,10.689,149.517
C02910=1110.830,322.790,-81.084,-177.603,10.692,149.517
C02911=1110.827,323.002,-81.113,-177.600,10.694,149.517
C02912=1110.824,323.214,-81.141,-177.598,10.695,149.517
C02913=1110.820,323.426,-81.170,-177.595,10.698,149.517
C02914=1110.817,323.638,-81.199,-177.592,10.700,149.517
C02915=1110.813,323.850,-81.227,-177.590,10.702,149.516
C02916=1110.810,324.063,-81.256,-177.587,10.705,149.516
C02917=1110.806,324.310,-81.290,-177.584,10.707,149.516
C02918=1110.802,324.558,-81.323,-177.580,10.710,149.516
C02919=1110.797,324.805,-81.356,-177.578,10.712,149.516
C02920=1110.794,325.053,-81.391,-177.575,10.714,149.515
C02921=1110.790,325.301,-81.424,-177.571,10.716,149.515
C02922=1110.786,325.549,-81.457,-177.568,10.719,149.515
C02923=1110.782,325.796,-81.491,-177.565,10.722,149.515
C02924=1110.778,326.044,-81.524,-177.562,10.724,149.515
C02925=1110.774,326.292,-81.558,-177.559,10.727,149.515
C02926=1110.770,326.539,-81.592,-177.555,10.729,149.514
C02927=1110.766,326.787,-81.625,-177.553,10.732,149.514
C02928=1110.762,327.034,-81.659,-177.549,10.735,149.514
C02929=1110.758,327.283,-81.693,-177.547,10.736,149.514
C02930=1110.754,327.530,-81.726,-177.544,10.739,149.514
C02931=1110.750,327.777,-81.760,-177.540,10.741,149.513
C02932=1110.746,328.026,-81.794,-177.537,10.744,149.513
C02933=1110.742,328.273,-81.828,-177.534,10.747,149.513
C02934=1110.738,328.520,-81.861,-177.531,10.749,149.513
C02935=1110.734,328.768,-81.895,-177.527,10.752,149.513
C02936=1110.730,329.016,-81.929,-177.524,10.754,149.512
C02937=1110.726,329.264,-81.963,-177.521,10.757,149.512
C02938=1110.722,329.511,-81.996,-177.518,10.759,149.512
C02939=1110.719,329.760,-82.030,-177.515,10.761,149.512
C02940=1110.714,330.007,-82.064,-177.512,10.764,149.512
C02941=1110.710,330.254,-82.098,-177.509,10.766,149.512
C02942=1110.707,330.503,-82.132,-177.506,10.769,149.511
C02943=1110.702,330.750,-82.166,-177.503,10.771,149.511
C02944=1110.698,330.997,-82.200,-177.499,10.774,149.511
C02945=1110.695,331.245,-82.234,-177.496,10.776,149.511
C02946=1110.691,331.493,-82.268,-177.493,10.779,149.511
C02947=1110.686,331.740,-82.302,-177.490,10.782,149.511
C02948=1110.683,331.988,-82.336,-177.486,10.784,149.510
C02949=1110.679,332.236,-82.369,-177.484,10.786,149.510
C02950=1110.675,332.484,-82.404,-177.481,10.788,149.510
C02951=1110.671,332.731,-82.438,-177.478,10.791,149.510
C02952=1110.667,332.978,-82.473,-177.474,10.793,149.509
C02953=1110.663,333.227,-82.506,-177.471,10.796,149.509
C02954=1110.659,333.474,-82.540,-177.468,10.799,149.509
C02955=1110.655,333.722,-82.575,-177.465,10.801,149.509
C02956=1110.652,333.969,-82.609,-177.462,10.804,149.509
C02957=1110.647,334.216,-82.643,-177.458,10.806,149.509
C02958=1110.644,334.464,-82.677,-177.455,10.809,149.508
C02959=1110.640,334.712,-82.711,-177.452,10.810,149.508
C02960=1110.636,334.960,-82.745,-177.450,10.813,149.508
C02961=1110.632,335.207,-82.779,-177.446,10.816,149.508
C02962=1110.628,335.455,-82.814,-177.443,10.818,149.508
C02963=1110.624,335.702,-82.848,-177.440,10.821,149.507
C02964=1110.620,335.951,-82.883,-177.437,10.823,149.507
C02965=1110.616,336.162,-82.912,-177.434,10.825,149.507
C02966=1110.614,336.374,-82.941,-177.431,10.828,149.507
C02967=1110.610,336.586,-82.970,-177.428,10.829,149.507
C02968=1110.607,336.798,-83.000,-177.426,10.831,149.507
C02969=1110.604,337.010,-83.029,-177.423,10.834,149.506
C02970=1110.600,337.222,-83.059,-177.420,10.836,149.506
C02971=1110.597,337.434,-83.088,-177.418,10.838,149.506
C02972=1110.593,337.646,-83.118,-177.415,10.840,149.506
C02973=1110.589,337.893,-83.152,-177.412,10.843,149.506
C02974=1110.585,338.141,-83.187,-177.409,10.845,149.506
C02975=1110.581,338.388,-83.222,-177.406,10.847,149.505
C02976=1110.578,338.636,-83.256,-177.403,10.850,149.505
C02977=1110.573,338.883,-83.290,-177.399,10.852,149.505
C02978=1110.570,339.131,-83.325,-177.396,10.855,149.505
C02979=1110.566,339.379,-83.359,-177.393,10.857,149.505
C02980=1110.562,339.627,-83.394,-177.390,10.860,149.504
C02981=1110.558,339.874,-83.428,-177.386,10.862,149.504
C02982=1110.554,340.121,-83.463,-177.383,10.865,149.504
C02983=1110.550,340.369,-83.498,-177.380,10.867,149.504
C02984=1110.546,340.617,-83.532,-177.378,10.869,149.504
C02985=1110.542,340.864,-83.567,-177.374,10.872,149.503
C02986=1110.538,341.112,-83.601,-177.371,10.874,149.503
C02987=1110.534,341.359,-83.636,-177.368,10.877,149.503
C02988=1110.530,341.607,-83.671,-177.365,10.879,149.503
C02989=1110.526,341.854,-83.705,-177.361,10.882,149.503
C02990=1110.523,342.101,-83.740,-177.358,10.884,149.502
C02991=1110.519,342.349,-83.775,-177.355,10.887,149.502
C02992=1110.514,342.597,-83.810,-177.351,10.889,149.502
C02993=1110.511,342.844,-83.845,-177.349,10.891,149.502
C02994=1110.507,343.091,-83.879,-177.346,10.894,149.502
C02995=1110.503,343.340,-83.914,-177.342,10.896,149.501
C02996=1110.499,343.587,-83.949,-177.339,10.899,149.501
C02997=1110.495,343.834,-83.984,-177.336,10.901,149.501
C02998=1110.492,344.082,-84.019,-177.333,10.904,149.501
C02999=1110.488,344.330,-84.054,-177.330,10.906,149.501
C03000=1110.483,344.577,-84.088,-177.326,10.909,149.501
C03001=1110.479,344.825,-84.124,-177.323,10.911,149.500
C03002=1110.475,345.072,-84.158,-177.320,10.914,149.500
C03003=1110.472,345.319,-84.193,-177.317,10.916,149.500
C03004=1110.468,345.567,-84.228,-177.314,10.918,149.500
C03005=1110.464,345.814,-84.263,-177.311,10.921,149.500
C03006=1110.460,346.062,-84.298,-177.307,10.923,149.499
C03007=1110.456,346.310,-84.333,-177.304,10.926,149.499
C03008=1110.452,346.557,-84.369,-177.301,10.928,149.499
C03009=1110.448,346.805,-84.403,-177.298,10.931,149.499
C03010=1110.445,347.052,-84.438,-177.295,10.933,149.499
C03011=1110.440,347.299,-84.473,-177.291,10.936,149.498
C03012=1110.437,347.547,-84.508,-177.288,10.938,149.498
C03013=1110.433,347.794,-84.544,-177.285,10.940,149.498
C03014=1110.429,348.043,-84.579,-177.282,10.943,149.498
C03015=1110.425,348.289,-84.614,-177.279,10.945,149.498
C03016=1110.421,348.537,-84.650,-177.276,10.948,149.497
C03017=1110.417,348.785,-84.684,-177.272,10.950,149.497
C03018=1110.413,349.032,-84.720,-177.269,10.953,149.497
C03019=1110.409,349.279,-84.755,-177.266,10.955,149.497
C03020=1110.405,349.527,-84.790,-177.263,10.958,149.497
C03021=1110.402,349.739,-84.820,-177.260,10.959,149.496
C03022=1110.399,349.951,-84.851,-177.257,10.962,149.496
C03023=1110.395,350.162,-84.881,-177.255,10.964,149.496
C03024=1110.392,350.374,-84.911,-177.252,10.966,149.496
C03025=1110.389,350.586,-84.941,-177.249,10.968,149.496
C03026=1110.386,350.797,-84.971,-177.246,10.970,149.496
C03027=1110.382,351.010,-85.002,-177.243,10.973,149.495
C03028=1110.379,351.222,-85.032,-177.240,10.974,149.495
C03029=1110.376,351.469,-85.067,-177.237,10.977,149.495
C03030=1110.371,351.716,-85.103,-177.234,10.979,149.495
C03031=1110.368,351.963,-85.138,-177.230,10.982,149.494
C03032=1110.364,352.211,-85.174,-177.227,10.984,149.494
C03033=1110.360,352.458,-85.209,-177.224,10.987,149.494
C03034=1110.356,352.706,-85.244,-177.221,10.989,149.494
C03035=1110.352,352.953,-85.279,-177.217,10.992,149.493
C03036=1110.349,353.201,-85.315,-177.214,10.994,149.493
C03037=1110.344,353.449,-85.351,-177.211,10.996,149.493
C03038=1110.340,353.696,-85.386,-177.207,10.999,149.493
C03039=1110.337,353.944,-85.422,-177.204,11.001,149.493
C03040=1110.333,354.191,-85.458,-177.201,11.004,149.492
C03041=1110.329,354.438,-85.493,-177.197,11.006,149.492
C03042=1110.325,354.685,-85.528,-177.194,11.008,149.492
C03043=1110.322,354.932,-85.565,-177.190,11.011,149.492
C03044=1110.318,355.180,-85.600,-177.187,11.013,149.491
C03045=1110.314,355.428,-85.636,-177.184,11.016,149.491
C03046=1110.310,355.675,-85.672,-177.180,11.018,149.491
C03047=1110.307,355.923,-85.707,-177.177,11.021,149.491
C03048=1110.303,356.170,-85.743,-177.174,11.023,149.490
C03049=1110.299,356.418,-85.778,-177.171,11.026,149.490
C03050=1110.295,356.665,-85.815,-177.167,11.028,149.490
C03051=1110.291,356.912,-85.850,-177.164,11.030,149.490
C03052=1110.287,357.159,-85.886,-177.160,11.033,149.489
C03053=1110.283,357.407,-85.922,-177.157,11.035,149.489
C03054=1110.280,357.654,-85.957,-177.154,11.038,149.489
C03055=1110.275,357.902,-85.993,-177.150,11.040,149.489
C03056=1110.272,358.149,-86.030,-177.147,11.042,149.488
C03057=1110.268,358.396,-86.065,-177.143,11.045,149.488
C03058=1110.265,358.644,-86.101,-177.140,11.047,149.488
C03059=1110.261,358.891,-86.137,-177.137,11.050,149.488
C03060=1110.257,359.138,-86.173,-177.133,11.052,149.487
C03061=1110.253,359.386,-86.209,-177.130,11.055,149.487
C03062=1110.249,359.633,-86.245,-177.126,11.057,149.487
C03063=1110.246,359.881,-86.281,-177.124,11.058,149.487
C03064=1110.242,360.128,-86.317,-177.120,11.061,149.486
C03065=1110.238,360.375,-86.353,-177.117,11.063,149.486
C03066=1110.234,360.623,-86.389,-177.114,11.066,149.486
C03067=1110.231,360.870,-86.425,-177.110,11.068,149.485
C03068=1110.226,361.118,-86.461,-177.107,11.070,149.485
C03069=1110.223,361.365,-86.497,-177.103,11.073,149.485
C03070=1110.219,361.612,-86.533,-177.100,11.075,149.485
C03071=1110.215,361.860,-86.569,-177.096,11.078,149.484
C03072=1110.212,362.107,-86.606,-177.093,11.080,149.484
C03073=1110.208,362.354,-86.641,-177.090,11.083,149.484
C03074=1110.204,362.601,-86.678,-177.087,11.085,149.484
C03075=1110.200,362.849,-86.714,-177.083,11.087,149.484
C03076=1110.196,363.096,-86.750,-177.080,11.090,149.483
C03077=1110.193,363.308,-86.781,-177.077,11.092,149.483
C03078=1110.190,363.520,-86.813,-177.074,11.094,149.483
C03079=1110.187,363.732,-86.844,-177.071,11.096,149.483
C03080=1110.184,363.943,-86.875,-177.068,11.098,149.482
C03081=1110.181,364.154,-86.906,-177.065,11.100,149.482
C03082=1110.177,364.366,-86.936,-177.062,11.102,149.482
C03083=1110.174,364.577,-86.967,-177.059,11.104,149.482
C03084=1110.171,364.789,-86.998,-177.057,11.106,149.481
C03085=1110.167,365.037,-87.035,-177.053,11.108,149.481
C03086=1110.163,365.283,-87.072,-177.050,11.111,149.481
C03087=1110.159,365.531,-87.108,-177.047,11.113,149.481
C03088=1110.155,365.778,-87.144,-177.043,11.115,149.480
C03089=1110.152,366.026,-87.181,-177.040,11.118,149.480
C03090=1110.149,366.273,-87.217,-177.036,11.120,149.480
C03091=1110.144,366.521,-87.254,-177.033,11.123,149.480
C03092=1110.140,366.768,-87.290,-177.030,11.125,149.480
C03093=1110.137,367.015,-87.327,-177.026,11.127,149.479
C03094=1110.133,367.262,-87.364,-177.023,11.130,149.479
C03095=1110.129,367.509,-87.400,-177.020,11.132,149.479
C03096=1110.126,367.757,-87.436,-177.016,11.135,149.479
C03097=1110.121,368.005,-87.473,-177.013,11.137,149.478
C03098=1110.118,368.251,-87.509,-177.009,11.139,149.478
C03099=1110.114,368.499,-87.546,-177.006,11.142,149.478
C03100=1110.111,368.745,-87.583,-177.003,11.144,149.478
C03101=1110.107,368.993,-87.619,-176.999,11.147,149.477
C03102=1110.103,369.241,-87.657,-176.996,11.149,149.477
C03103=1110.100,369.487,-87.693,-176.993,11.152,149.477
C03104=1110.096,369.735,-87.730,-176.989,11.154,149.477
C03105=1110.091,369.982,-87.767,-176.986,11.156,149.476
C03106=1110.087,370.229,-87.803,-176.982,11.159,149.476
C03107=1110.085,370.477,-87.840,-176.979,11.161,149.476
C03108=1110.081,370.724,-87.877,-176.975,11.165,149.476
C03109=1110.076,370.971,-87.914,-176.972,11.167,149.476
C03110=1110.073,371.218,-87.950,-176.969,11.170,149.475
C03111=1110.070,371.466,-87.987,-176.965,11.172,149.475
C03112=1110.066,371.713,-88.024,-176.962,11.174,149.475
C03113=1110.061,371.960,-88.061,-176.958,11.177,149.475
C03114=1110.058,372.207,-88.097,-176.955,11.179,149.474
C03115=1110.055,372.455,-88.134,-176.952,11.182,149.474
C03116=1110.050,372.702,-88.171,-176.948,11.184,149.474
C03117=1110.046,372.949,-88.208,-176.945,11.187,149.474
C03118=1110.042,373.196,-88.245,-176.942,11.189,149.474
C03119=1110.040,373.443,-88.282,-176.939,11.192,149.473
C03120=1110.036,373.691,-88.319,-176.935,11.194,149.473
C03121=1110.032,373.938,-88.356,-176.932,11.196,149.473
C03122=1110.028,374.186,-88.393,-176.928,11.199,149.473
C03123=1110.024,374.432,-88.431,-176.925,11.201,149.472
C03124=1110.020,374.679,-88.468,-176.922,11.204,149.472
C03125=1110.018,374.927,-88.504,-176.918,11.206,149.472
C03126=1110.013,375.174,-88.541,-176.915,11.209,149.472
C03127=1110.010,375.421,-88.579,-176.911,11.212,149.472
C03128=1110.006,375.669,-88.616,-176.908,11.214,149.471
C03129=1110.002,375.916,-88.653,-176.905,11.217,149.471
C03130=1109.998,376.162,-88.691,-176.901,11.219,149.471
C03131=1109.995,376.410,-88.728,-176.898,11.222,149.471
C03132=1109.991,376.658,-88.765,-176.895,11.224,149.471
C03133=1109.987,376.909,-88.803,-176.891,11.227,149.470
C03134=1109.984,377.160,-88.841,-176.888,11.229,149.470
C03135=1109.980,377.412,-88.879,-176.884,11.233,149.470
C03136=1109.976,377.664,-88.917,-176.881,11.235,149.470
C03137=1109.972,377.911,-88.954,-176.878,11.238,149.470
C03138=1109.968,378.157,-88.991,-176.875,11.240,149.470
C03139=1109.965,378.405,-89.028,-176.871,11.243,149.469
C03140=1109.961,378.652,-89.066,-176.868,11.245,149.469
C03141=1109.957,378.900,-89.103,-176.865,11.248,149.469
C03142=1109.954,379.146,-89.141,-176.861,11.251,149.469
C03143=1109.949,379.393,-89.178,-176.858,11.254,149.469
C03144=1109.946,379.641,-89.216,-176.854,11.256,149.468
C03145=1109.942,379.888,-89.252,-176.851,11.259,149.468
C03146=1109.939,380.135,-89.290,-176.848,11.261,149.468
C03147=1109.935,380.382,-89.328,-176.845,11.264,149.468
C03148=1109.932,380.630,-89.365,-176.841,11.267,149.468
C03149=1109.928,380.876,-89.403,-176.838,11.270,149.468
C03150=1109.923,381.123,-89.441,-176.835,11.272,149.468
C03151=1109.920,381.371,-89.478,-176.831,11.275,149.468
C03152=1109.916,381.618,-89.516,-176.828,11.277,149.467
C03153=1109.913,381.865,-89.554,-176.825,11.280,149.467
C03154=1109.909,382.112,-89.590,-176.821,11.284,149.467
C03155=1109.906,382.359,-89.628,-176.818,11.286,149.467
C03156=1109.902,382.606,-89.666,-176.815,11.289,149.467
C03157=1109.898,382.854,-89.703,-176.812,11.291,149.467
C03158=1109.894,383.101,-89.741,-176.809,11.294,149.467
C03159=1109.891,383.348,-89.779,-176.805,11.297,149.466
C03160=1109.887,383.594,-89.817,-176.802,11.300,149.466
C03161=1109.884,383.842,-89.855,-176.799,11.302,149.466
C03162=1109.880,384.089,-89.892,-176.797,11.305,149.466
C03163=1109.876,384.337,-89.930,-176.793,11.307,149.466
C03164=1109.872,384.583,-89.968,-176.790,11.310,149.466
C03165=1109.869,384.830,-90.006,-176.788,11.313,149.466
C03166=1109.865,385.078,-90.044,-176.785,11.315,149.466
C03167=1109.862,385.324,-90.081,-176.782,11.318,149.466
C03168=1109.858,385.572,-90.120,-176.779,11.321,149.466
C03169=1109.854,385.818,-90.157,-176.777,11.323,149.466
C03170=1109.851,386.066,-90.195,-176.774,11.326,149.466
C03171=1109.847,386.312,-90.233,-176.771,11.329,149.466
C03172=1109.843,386.560,-90.271,-176.768,11.332,149.466
C03173=1109.590,375.445,-88.642,-176.911,11.213,149.472
C03174=1109.593,375.197,-88.605,-176.914,11.210,149.472
C03175=1109.597,374.951,-88.568,-176.917,11.208,149.472
C03176=1109.601,374.704,-88.531,-176.921,11.205,149.472
C03177=1109.604,374.456,-88.494,-176.924,11.202,149.472
C03178=1109.609,374.208,-88.457,-176.928,11.200,149.473
C03179=1109.612,373.962,-88.420,-176.931,11.197,149.473
C03180=1109.615,373.714,-88.383,-176.934,11.195,149.473
C03181=1109.619,373.467,-88.346,-176.938,11.192,149.473
C03182=1109.623,373.220,-88.309,-176.941,11.190,149.473
C03183=1109.627,372.973,-88.272,-176.944,11.187,149.474
C03184=1109.630,372.725,-88.235,-176.947,11.185,149.474
C03185=1109.634,372.479,-88.198,-176.951,11.182,149.474
C03186=1109.638,372.231,-88.161,-176.954,11.180,149.474
C03187=1109.642,371.983,-88.124,-176.957,11.177,149.474
C03188=1109.646,371.736,-88.087,-176.961,11.175,149.475
C03189=1109.649,371.489,-88.051,-176.964,11.173,149.475
C03190=1109.653,371.242,-88.014,-176.968,11.170,149.475
C03191=1109.657,370.994,-87.976,-176.971,11.168,149.475
C03192=1109.660,370.747,-87.940,-176.974,11.165,149.476
C03193=1109.664,370.500,-87.903,-176.978,11.162,149.476
C03194=1109.668,370.253,-87.866,-176.981,11.159,149.476
C03195=1109.672,370.006,-87.830,-176.985,11.157,149.476
C03196=1109.675,369.758,-87.793,-176.988,11.155,149.477
C03197=1109.679,369.511,-87.756,-176.992,11.152,149.477
C03198=1109.683,369.264,-87.719,-176.995,11.150,149.477
C03199=1109.687,369.017,-87.683,-176.998,11.147,149.477
C03200=1109.691,368.770,-87.646,-177.002,11.145,149.477
C03201=1109.694,368.522,-87.609,-177.005,11.143,149.478
C03202=1109.697,368.275,-87.573,-177.009,11.140,149.478
C03203=1109.702,368.027,-87.537,-177.012,11.138,149.478
C03204=1109.706,367.780,-87.500,-177.015,11.135,149.478
C03205=1109.709,367.533,-87.463,-177.019,11.133,149.479
C03206=1109.713,367.286,-87.427,-177.022,11.131,149.479
C03207=1109.716,367.038,-87.390,-177.026,11.128,149.479
C03208=1109.720,366.791,-87.353,-177.029,11.126,149.479
C03209=1109.724,366.544,-87.317,-177.032,11.123,149.480
C03210=1109.728,366.297,-87.281,-177.035,11.121,149.480
C03211=1109.732,366.049,-87.244,-177.039,11.119,149.480
C03212=1109.735,365.802,-87.208,-177.042,11.116,149.480
C03213=1109.740,365.555,-87.171,-177.046,11.114,149.481
C03214=1109.743,365.308,-87.135,-177.049,11.111,149.481
C03215=1109.747,365.061,-87.098,-177.052,11.109,149.481
C03216=1109.750,364.812,-87.062,-177.056,11.107,149.482
C03217=1109.754,364.565,-87.025,-177.059,11.104,149.482
C03218=1109.760,364.199,-86.972,-177.064,11.100,149.482
C03219=1109.766,363.831,-86.918,-177.069,11.097,149.482
C03220=1109.771,363.464,-86.864,-177.074,11.094,149.483
C03221=1109.776,363.097,-86.810,-177.079,11.090,149.483
C03222=1109.781,362.849,-86.774,-177.082,11.088,149.483
C03223=1109.784,362.602,-86.738,-177.086,11.085,149.484
C03224=1109.788,362.355,-86.702,-177.089,11.083,149.484
C03225=1109.792,362.107,-86.665,-177.093,11.081,149.484
C03226=1109.796,361.860,-86.630,-177.096,11.078,149.484
C03227=1109.800,361.613,-86.593,-177.099,11.076,149.485
C03228=1109.803,361.365,-86.557,-177.103,11.074,149.485
C03229=1109.807,361.118,-86.521,-177.106,11.071,149.485
C03230=1109.811,360.871,-86.485,-177.109,11.069,149.486
C03231=1109.814,360.624,-86.449,-177.113,11.066,149.486
C03232=1109.818,360.376,-86.413,-177.116,11.064,149.486
C03233=1109.822,360.128,-86.377,-177.120,11.062,149.486
C03234=1109.826,359.881,-86.341,-177.123,11.059,149.487
C03235=1109.830,359.634,-86.305,-177.126,11.057,149.487
C03236=1109.834,359.387,-86.268,-177.130,11.054,149.487
C03237=1109.837,359.139,-86.233,-177.133,11.052,149.487
C03238=1109.841,358.892,-86.197,-177.137,11.050,149.488
C03239=1109.844,358.645,-86.161,-177.140,11.047,149.488
C03240=1109.849,358.397,-86.125,-177.143,11.045,149.488
C03241=1109.852,358.150,-86.089,-177.147,11.042,149.488
C03242=1109.856,357.902,-86.054,-177.150,11.040,149.489
C03243=1109.860,357.655,-86.017,-177.153,11.037,149.489
C03244=1109.864,357.407,-85.981,-177.157,11.035,149.489
C03245=1109.867,357.160,-85.946,-177.160,11.033,149.489
C03246=1109.871,356.912,-85.910,-177.164,11.030,149.490
C03247=1109.875,356.666,-85.875,-177.167,11.028,149.490
C03248=1109.879,356.418,-85.838,-177.170,11.025,149.490
C03249=1109.883,356.171,-85.803,-177.173,11.023,149.490
C03250=1109.887,355.923,-85.767,-177.176,11.021,149.490
C03251=1109.890,355.676,-85.731,-177.180,11.019,149.491
C03252=1109.894,355.428,-85.696,-177.183,11.017,149.491
C03253=1109.899,355.181,-85.660,-177.186,11.014,149.491
C03254=1109.902,354.933,-85.624,-177.190,11.012,149.492
C03255=1109.906,354.686,-85.589,-177.193,11.009,149.492
C03256=1109.910,354.439,-85.553,-177.196,11.007,149.492
C03257=1109.914,354.191,-85.518,-177.200,11.004,149.492
C03258=1109.917,353.944,-85.482,-177.203,11.002,149.492
C03259=1109.921,353.696,-85.447,-177.206,10.999,149.493
C03260=1109.925,353.449,-85.411,-177.210,10.997,149.493
C03261=1109.929,353.201,-85.375,-177.213,10.994,149.493
C03262=1109.933,352.953,-85.340,-177.217,10.992,149.494
C03263=1109.937,352.707,-85.304,-177.220,10.990,149.494
C03264=1109.941,352.459,-85.269,-177.223,10.987,149.494
C03265=1109.944,352.212,-85.233,-177.227,10.985,149.494
C03266=1109.948,351.964,-85.198,-177.230,10.982,149.494
C03267=1109.952,351.717,-85.162,-177.233,10.980,149.495
C03268=1109.956,351.470,-85.127,-177.236,10.978,149.495
C03269=1109.960,351.222,-85.091,-177.240,10.975,149.495
C03270=1109.963,351.010,-85.062,-177.243,10.972,149.495
C03271=1109.967,350.798,-85.031,-177.245,10.971,149.495
C03272=1109.969,350.587,-85.001,-177.248,10.969,149.496
C03273=1109.972,350.375,-84.970,-177.251,10.966,149.496
C03274=1109.976,350.163,-84.941,-177.254,10.964,149.496
C03275=1109.980,349.951,-84.910,-177.257,10.962,149.496
C03276=1109.983,349.740,-84.880,-177.259,10.960,149.496
C03277=1109.986,349.528,-84.850,-177.263,10.957,149.496
C03278=1109.990,349.280,-84.815,-177.265,10.956,149.497
C03279=1109.994,349.033,-84.780,-177.269,10.953,149.497
C03280=1109.997,348.786,-84.744,-177.272,10.951,149.497
C03281=1110.001,348.538,-84.709,-177.275,10.948,149.497
C03282=1110.005,348.290,-84.674,-177.278,10.946,149.497
C03283=1110.009,348.043,-84.638,-177.281,10.943,149.498
C03284=1110.013,347.795,-84.604,-177.285,10.941,149.498
C03285=1110.017,347.548,-84.568,-177.288,10.938,149.498
C03286=1110.021,347.301,-84.533,-177.291,10.936,149.498
C03287=1110.025,347.053,-84.499,-177.294,10.934,149.498
C03288=1110.028,346.806,-84.463,-177.297,10.931,149.499
C03289=1110.033,346.558,-84.429,-177.300,10.929,149.499
C03290=1110.036,346.311,-84.393,-177.304,10.926,149.499
C03291=1110.040,346.063,-84.358,-177.307,10.924,149.499
C03292=1110.045,345.816,-84.323,-177.310,10.921,149.500
C03293=1110.048,345.568,-84.288,-177.313,10.919,149.500
C03294=1110.052,345.320,-84.253,-177.316,10.916,149.500
C03295=1110.056,345.074,-84.218,-177.320,10.914,149.500
C03296=1110.060,344.826,-84.183,-177.323,10.911,149.500
C03297=1110.063,344.578,-84.148,-177.326,10.910,149.501
C03298=1110.068,344.331,-84.113,-177.329,10.907,149.501
C03299=1110.071,344.083,-84.079,-177.332,10.904,149.501
C03300=1110.075,343.835,-84.043,-177.335,10.902,149.501
C03301=1110.079,343.588,-84.009,-177.339,10.899,149.501
C03302=1110.083,343.340,-83.973,-177.342,10.897,149.502
C03303=1110.088,343.093,-83.939,-177.345,10.894,149.502
C03304=1110.091,342.845,-83.905,-177.348,10.892,149.502
C03305=1110.095,342.598,-83.869,-177.351,10.889,149.502
C03306=1110.099,342.350,-83.835,-177.354,10.888,149.502
C03307=1110.103,342.102,-83.800,-177.357,10.885,149.502
C03308=1110.107,341.856,-83.765,-177.360,10.882,149.503
C03309=1110.111,341.608,-83.730,-177.364,10.880,149.503
C03310=1110.115,341.359,-83.696,-177.367,10.877,149.503
C03311=1110.118,341.113,-83.661,-177.370,10.875,149.503
C03312=1110.122,340.865,-83.626,-177.373,10.872,149.503
C03313=1110.127,340.617,-83.592,-177.376,10.870,149.504
C03314=1110.130,340.370,-83.558,-177.380,10.867,149.504
C03315=1110.134,340.123,-83.522,-177.383,10.865,149.504
C03316=1110.138,339.875,-83.488,-177.385,10.863,149.504
C03317=1110.142,339.628,-83.454,-177.389,10.860,149.504
C03318=1110.146,339.379,-83.419,-177.392,10.858,149.505
C03319=1110.150,339.132,-83.384,-177.395,10.855,149.505
C03320=1110.154,338.884,-83.350,-177.398,10.853,149.505
C03321=1110.158,338.637,-83.316,-177.402,10.850,149.505
C03322=1110.161,338.390,-83.281,-177.405,10.848,149.505
C03323=1110.166,338.142,-83.246,-177.408,10.845,149.506
C03324=1110.170,337.894,-83.211,-177.411,10.843,149.506
C03325=1110.174,337.647,-83.178,-177.414,10.840,149.506
C03326=1110.177,337.435,-83.148,-177.417,10.838,149.506
C03327=1110.180,337.222,-83.118,-177.419,10.836,149.506
C03328=1110.184,337.011,-83.089,-177.423,10.834,149.506
C03329=1110.187,336.799,-83.059,-177.425,10.832,149.507
C03330=1110.191,336.587,-83.030,-177.428,10.830,149.507
C03331=1110.193,336.375,-83.001,-177.431,10.827,149.507
C03332=1110.197,336.163,-82.972,-177.433,10.826,149.507
C03333=1110.200,335.951,-82.942,-177.436,10.824,149.507
C03334=1110.204,335.703,-82.908,-177.439,10.821,149.507
C03335=1110.208,335.456,-82.874,-177.442,10.819,149.508
C03336=1110.212,335.208,-82.839,-177.445,10.816,149.508
C03337=1110.216,334.961,-82.805,-177.448,10.814,149.508
C03338=1110.220,334.714,-82.771,-177.452,10.811,149.508
C03339=1110.224,334.466,-82.736,-177.455,10.808,149.508
C03340=1110.228,334.219,-82.702,-177.458,10.806,149.508
C03341=1110.232,333.970,-82.668,-177.461,10.804,149.509
C03342=1110.236,333.723,-82.634,-177.464,10.802,149.509
C03343=1110.240,333.475,-82.600,-177.467,10.799,149.509
C03344=1110.243,333.227,-82.566,-177.470,10.797,149.509
C03345=1110.247,332.980,-82.532,-177.474,10.794,149.510
C03346=1110.252,332.732,-82.498,-177.477,10.791,149.510
C03347=1110.255,332.485,-82.464,-177.480,10.789,149.510
C03348=1110.259,332.237,-82.430,-177.483,10.786,149.510
C03349=1110.263,331.989,-82.395,-177.486,10.784,149.510
C03350=1110.267,331.742,-82.361,-177.489,10.781,149.510
C03351=1110.271,331.494,-82.328,-177.492,10.780,149.511
C03352=1110.275,331.246,-82.293,-177.495,10.777,149.511
C03353=1110.279,330.999,-82.259,-177.498,10.774,149.511
C03354=1110.283,330.751,-82.226,-177.502,10.772,149.511
C03355=1110.287,330.503,-82.191,-177.505,10.769,149.511
C03356=1110.291,330.256,-82.158,-177.508,10.767,149.511
C03357=1110.294,330.008,-82.124,-177.511,10.764,149.512
C03358=1110.299,329.760,-82.090,-177.515,10.762,149.512
C03359=1110.303,329.513,-82.056,-177.517,10.759,149.512
C03360=1110.306,329.265,-82.022,-177.521,10.756,149.512
C03361=1110.310,329.018,-81.988,-177.523,10.755,149.513
C03362=1110.315,328.770,-81.955,-177.527,10.752,149.513
C03363=1110.318,328.522,-81.920,-177.530,10.750,149.513
C03364=1110.322,328.274,-81.887,-177.533,10.747,149.513
C03365=1110.326,328.027,-81.853,-177.536,10.745,149.513
C03366=1110.330,327.779,-81.820,-177.539,10.742,149.513
C03367=1110.334,327.531,-81.785,-177.543,10.739,149.514
C03368=1110.339,327.283,-81.752,-177.546,10.737,149.514
C03369=1110.342,327.036,-81.718,-177.549,10.734,149.514
C03370=1110.346,326.788,-81.685,-177.552,10.732,149.514
C03371=1110.350,326.541,-81.651,-177.555,10.730,149.514
C03372=1110.355,326.293,-81.617,-177.558,10.727,149.514
C03373=1110.359,326.045,-81.584,-177.561,10.725,149.515
C03374=1110.362,325.797,-81.550,-177.564,10.722,149.515
C03375=1110.366,325.550,-81.517,-177.567,10.720,149.515
C03376=1110.370,325.302,-81.483,-177.571,10.717,149.515
C03377=1110.374,325.055,-81.450,-177.574,10.714,149.515
C03378=1110.378,324.806,-81.416,-177.577,10.712,149.516
C03379=1110.381,324.559,-81.382,-177.580,10.710,149.516
C03380=1110.386,324.311,-81.349,-177.582,10.708,149.516
C03381=1110.390,324.064,-81.316,-177.586,10.705,149.516
C03382=1110.393,323.851,-81.286,-177.589,10.702,149.516
C03383=1110.396,323.640,-81.258,-177.591,10.701,149.516
C03384=1110.400,323.427,-81.230,-177.594,10.699,149.517
C03385=1110.403,323.215,-81.201,-177.597,10.696,149.517
C03386=1110.407,323.003,-81.172,-177.599,10.694,149.517
C03387=1110.410,322.791,-81.144,-177.602,10.692,149.517
C03388=1110.414,322.579,-81.115,-177.605,10.690,149.517
C03389=1110.417,322.367,-81.087,-177.607,10.688,149.517
C03390=1110.421,322.120,-81.054,-177.611,10.685,149.518
C03391=1110.425,321.871,-81.020,-177.614,10.683,149.518
C03392=1110.429,321.624,-80.986,-177.617,10.680,149.518
C03393=1110.433,321.376,-80.953,-177.620,10.678,149.518
C03394=1110.437,321.129,-80.920,-177.623,10.675,149.518
C03395=1110.441,320.881,-80.887,-177.626,10.673,149.519
C03396=1110.445,320.633,-80.854,-177.629,10.671,149.519
C03397=1110.449,320.385,-80.821,-177.632,10.668,149.519
C03398=1110.453,320.137,-80.787,-177.635,10.666,149.519
C03399=1110.457,319.889,-80.754,-177.639,10.663,149.519
C03400=1110.461,319.642,-80.721,-177.642,10.660,149.519
C03401=1110.465,319.394,-80.688,-177.645,10.658,149.520
C03402=1110.469,319.146,-80.655,-177.648,10.655,149.520
C03403=1110.473,318.899,-80.622,-177.651,10.653,149.520
C03404=1110.477,318.651,-80.589,-177.654,10.650,149.520
C03405=1110.481,318.403,-80.556,-177.657,10.648,149.520
C03406=1110.485,318.155,-80.522,-177.660,10.646,149.521
C03407=1110.489,317.907,-80.489,-177.663,10.643,149.521
C03408=1110.493,317.659,-80.456,-177.666,10.641,149.521
C03409=1110.496,317.412,-80.423,-177.670,10.638,149.521
C03410=1110.500,317.164,-80.390,-177.673,10.635,149.521
C03411=1110.504,316.916,-80.357,-177.676,10.633,149.521
C03412=1110.509,316.669,-80.324,-177.679,10.630,149.521
C03413=1110.513,316.421,-80.291,-177.682,10.628,149.522
C03414=1110.516,316.173,-80.259,-177.685,10.625,149.522
C03415=1110.521,315.925,-80.226,-177.688,10.623,149.522
C03416=1110.525,315.677,-80.192,-177.691,10.621,149.522
C03417=1110.529,315.430,-80.159,-177.694,10.618,149.522
C03418=1110.532,315.182,-80.127,-177.697,10.616,149.523
C03419=1110.537,314.934,-80.094,-177.700,10.613,149.523
C03420=1110.541,314.686,-80.061,-177.704,10.610,149.523
C03421=1110.545,314.439,-80.028,-177.707,10.608,149.523
C03422=1110.548,314.191,-79.995,-177.710,10.605,149.523
C03423=1110.553,313.943,-79.963,-177.713,10.603,149.524
C03424=1110.557,313.695,-79.930,-177.715,10.601,149.524
C03425=1110.560,313.448,-79.897,-177.719,10.598,149.524
C03426=1110.565,313.199,-79.865,-177.722,10.596,149.524
C03427=1110.569,312.952,-79.832,-177.725,10.593,149.524
C03428=1110.572,312.704,-79.799,-177.728,10.591,149.525
C03429=1110.577,312.456,-79.767,-177.731,10.588,149.525
C03430=1110.581,312.208,-79.733,-177.735,10.585,149.525
C03431=1110.584,311.961,-79.701,-177.738,10.583,149.525
C03432=1110.589,311.712,-79.668,-177.741,10.580,149.525
C03433=1110.593,311.465,-79.635,-177.744,10.577,149.525
C03434=1110.597,311.216,-79.603,-177.747,10.576,149.526
C03435=1110.601,310.969,-79.570,-177.750,10.573,149.526
C03436=1110.605,310.720,-79.538,-177.753,10.571,149.526
C03437=1110.609,310.474,-79.506,-177.756,10.568,149.526
C03438=1110.612,310.261,-79.477,-177.758,10.566,149.526
C03439=1110.616,310.049,-79.450,-177.761,10.563,149.526
C03440=1110.619,309.837,-79.422,-177.764,10.562,149.527
C03441=1110.623,309.625,-79.394,-177.766,10.560,149.527
C03442=1110.627,309.412,-79.366,-177.769,10.557,149.527
C03443=1110.630,309.200,-79.339,-177.772,10.555,149.527
C03444=1110.634,308.988,-79.311,-177.774,10.553,149.527
C03445=1110.637,308.775,-79.283,-177.777,10.550,149.527
C03446=1110.641,308.529,-79.251,-177.781,10.548,149.527
C03447=1110.645,308.280,-79.218,-177.783,10.545,149.528
C03448=1110.649,308.033,-79.186,-177.786,10.544,149.528
C03449=1110.653,307.784,-79.153,-177.789,10.541,149.528
C03450=1110.657,307.536,-79.122,-177.792,10.538,149.528
C03451=1110.661,307.289,-79.088,-177.796,10.536,149.528
C03452=1110.665,307.041,-79.057,-177.799,10.533,149.528
C03453=1110.670,306.793,-79.025,-177.802,10.531,149.529
C03454=1110.673,306.546,-78.992,-177.805,10.528,149.529
C03455=1110.677,306.297,-78.960,-177.808,10.526,149.529
C03456=1110.681,306.049,-78.928,-177.811,10.523,149.529
C03457=1110.686,305.801,-78.895,-177.815,10.520,149.529
C03458=1110.690,305.554,-78.863,-177.817,10.518,149.530
C03459=1110.694,305.306,-78.831,-177.820,10.516,149.530
C03460=1110.698,305.058,-78.799,-177.823,10.513,149.530
C03461=1110.701,304.810,-78.767,-177.826,10.511,149.530
C03462=1110.706,304.561,-78.734,-177.829,10.508,149.530
C03463=1110.710,304.315,-78.702,-177.833,10.506,149.530
C03464=1110.714,304.066,-78.670,-177.836,10.503,149.531
C03465=1110.718,303.818,-78.638,-177.839,10.500,149.531
C03466=1110.722,303.570,-78.606,-177.842,10.498,149.531
C03467=1110.727,303.323,-78.574,-177.845,10.496,149.531
C03468=1110.731,303.074,-78.542,-177.847,10.493,149.531
C03469=1110.734,302.826,-78.510,-177.851,10.491,149.532
C03470=1110.739,302.578,-78.478,-177.854,10.488,149.532
C03471=1110.743,302.331,-78.446,-177.857,10.485,149.532
C03472=1110.746,302.083,-78.414,-177.860,10.483,149.532
C03473=1110.751,301.835,-78.381,-177.863,10.480,149.532
C03474=1110.755,301.588,-78.350,-177.866,10.478,149.532
C03475=1110.759,301.340,-78.318,-177.870,10.475,149.533
C03476=1110.763,301.091,-78.286,-177.872,10.473,149.533
C03477=1110.767,300.843,-78.254,-177.875,10.471,149.533
C03478=1110.772,300.595,-78.223,-177.878,10.468,149.533
C03479=1110.775,300.347,-78.191,-177.881,10.465,149.533
C03480=1110.780,300.099,-78.159,-177.884,10.463,149.533
C03481=1110.784,299.852,-78.127,-177.888,10.460,149.534
C03482=1110.788,299.604,-78.095,-177.891,10.457,149.534
C03483=1110.791,299.355,-78.064,-177.894,10.455,149.534
C03484=1110.796,299.108,-78.032,-177.897,10.452,149.534
C03485=1110.800,298.860,-78.000,-177.900,10.450,149.534
C03486=1110.804,298.612,-77.968,-177.903,10.448,149.534
C03487=1110.808,298.364,-77.936,-177.906,10.445,149.535
C03488=1110.812,298.116,-77.905,-177.909,10.443,149.535
C03489=1110.816,297.868,-77.873,-177.912,10.440,149.535
C03490=1110.820,297.620,-77.842,-177.915,10.437,149.535
C03491=1110.825,297.372,-77.809,-177.918,10.435,149.535
C03492=1110.829,297.125,-77.778,-177.921,10.432,149.535
C03493=1110.833,296.876,-77.747,-177.925,10.430,149.536
C03494=1110.837,296.664,-77.720,-177.927,10.428,149.536
C03495=1110.840,296.451,-77.693,-177.929,10.426,149.536
C03496=1110.843,296.239,-77.666,-177.933,10.423,149.536
C03497=1110.847,296.026,-77.639,-177.935,10.421,149.536
C03498=1110.850,295.814,-77.612,-177.937,10.419,149.536
C03499=1110.854,295.602,-77.585,-177.940,10.417,149.536
C03500=1110.857,295.389,-77.558,-177.943,10.415,149.537
C03501=1110.861,295.178,-77.531,-177.945,10.413,149.537
C03502=1110.865,294.930,-77.500,-177.948,10.410,149.537
C03503=1110.868,294.682,-77.468,-177.951,10.408,149.537
C03504=1110.873,294.434,-77.437,-177.954,10.405,149.537
C03505=1110.877,294.186,-77.405,-177.958,10.403,149.538
C03506=1110.881,293.938,-77.374,-177.961,10.400,149.538
C03507=1110.885,293.690,-77.342,-177.964,10.397,149.538
C03508=1110.889,293.442,-77.311,-177.966,10.395,149.538
C03509=1110.893,293.194,-77.280,-177.970,10.393,149.538
C03510=1110.897,292.946,-77.248,-177.973,10.390,149.538
C03511=1110.902,292.698,-77.217,-177.976,10.388,149.539
C03512=1110.905,292.450,-77.185,-177.979,10.385,149.539
C03513=1110.910,292.202,-77.155,-177.982,10.382,149.539
C03514=1110.914,291.954,-77.123,-177.985,10.380,149.539
C03515=1110.918,291.706,-77.092,-177.988,10.377,149.539
C03516=1110.922,291.458,-77.060,-177.991,10.375,149.540
C03517=1110.927,291.210,-77.029,-177.994,10.373,149.540
C03518=1110.931,290.961,-76.998,-177.997,10.370,149.540
C03519=1110.935,290.714,-76.967,-178.000,10.368,149.540
C03520=1110.939,290.465,-76.936,-178.003,10.365,149.540
C03521=1110.942,290.218,-76.905,-178.006,10.362,149.540
C03522=1110.946,289.969,-76.874,-178.009,10.360,149.540
C03523=1110.951,289.721,-76.843,-178.012,10.357,149.541
C03524=1110.955,289.473,-76.811,-178.015,10.354,149.541
C03525=1110.959,289.225,-76.780,-178.019,10.352,149.541
C03526=1110.963,288.977,-76.749,-178.021,10.350,149.541
C03527=1110.968,288.729,-76.718,-178.024,10.348,149.541
C03528=1110.972,288.482,-76.688,-178.027,10.345,149.542
C03529=1110.976,288.233,-76.656,-178.031,10.342,149.542
C03530=1110.980,287.985,-76.626,-178.034,10.340,149.542
C03531=1110.984,287.737,-76.594,-178.037,10.337,149.542
C03532=1110.989,287.489,-76.563,-178.040,10.334,149.542
C03533=1110.992,287.241,-76.532,-178.043,10.332,149.542
C03534=1110.996,286.993,-76.502,-178.046,10.330,149.543
C03535=1111.001,286.745,-76.471,-178.048,10.327,149.543
C03536=1111.005,286.497,-76.439,-178.052,10.325,149.543
C03537=1111.009,286.249,-76.409,-178.055,10.322,149.543
C03538=1111.013,286.001,-76.378,-178.058,10.319,149.543
C03539=1111.017,285.753,-76.347,-178.061,10.317,149.543
C03540=1111.021,285.505,-76.317,-178.064,10.314,149.544
C03541=1111.025,285.256,-76.286,-178.067,10.312,149.544
C03542=1111.030,285.008,-76.255,-178.070,10.310,149.544
C03543=1111.034,284.760,-76.224,-178.073,10.307,149.544
C03544=1111.037,284.513,-76.193,-178.076,10.305,149.544
C03545=1111.042,284.265,-76.162,-178.079,10.302,149.544
C03546=1111.047,284.017,-76.131,-178.082,10.299,149.545
C03547=1111.050,283.768,-76.101,-178.085,10.297,149.545
C03548=1111.054,283.520,-76.070,-178.088,10.294,149.545
C03549=1111.059,283.273,-76.039,-178.091,10.291,149.545
C03550=1111.062,283.060,-76.013,-178.094,10.289,149.545
C03551=1111.066,282.847,-75.988,-178.096,10.287,149.545
C03552=1111.069,282.634,-75.960,-178.099,10.285,149.546
C03553=1111.073,282.422,-75.935,-178.102,10.283,149.546
C03554=1111.076,282.210,-75.909,-178.104,10.281,149.546
C03555=1111.079,281.997,-75.882,-178.107,10.278,149.546
C03556=1111.084,281.785,-75.856,-178.109,10.276,149.546
C03557=1111.087,281.572,-75.830,-178.112,10.275,149.546
C03558=1111.092,281.324,-75.800,-178.115,10.272,149.547
C03559=1111.095,281.076,-75.769,-178.118,10.269,149.547
C03560=1111.100,280.828,-75.738,-178.121,10.267,149.547
C03561=1111.104,280.580,-75.708,-178.124,10.264,149.547
C03562=1111.108,280.332,-75.677,-178.127,10.262,149.547
C03563=1111.112,280.083,-75.647,-178.130,10.259,149.547
C03564=1111.116,279.835,-75.617,-178.133,10.256,149.547
C03565=1111.120,279.588,-75.587,-178.137,10.254,149.548
C03566=1111.125,279.340,-75.556,-178.140,10.251,149.548
C03567=1111.129,279.092,-75.526,-178.142,10.249,149.548
C03568=1111.133,278.843,-75.495,-178.145,10.246,149.548
C03569=1111.137,278.595,-75.465,-178.148,10.244,149.548
C03570=1111.142,278.347,-75.434,-178.151,10.241,149.548
C03571=1111.146,278.099,-75.405,-178.154,10.238,149.549
C03572=1111.150,277.850,-75.374,-178.157,10.236,149.549
C03573=1111.154,277.603,-75.344,-178.160,10.233,149.549
C03574=1111.159,277.354,-75.313,-178.163,10.230,149.549
C03575=1111.162,277.107,-75.283,-178.166,10.227,149.549
C03576=1111.166,276.859,-75.253,-178.169,10.225,149.549
C03577=1111.171,276.610,-75.223,-178.172,10.222,149.549
C03578=1111.174,276.362,-75.193,-178.175,10.219,149.550
C03579=1111.179,276.114,-75.162,-178.178,10.217,149.550
C03580=1111.183,275.866,-75.132,-178.181,10.215,149.550
C03581=1111.187,275.618,-75.102,-178.184,10.212,149.550
C03582=1111.191,275.369,-75.072,-178.187,10.210,149.550
C03583=1111.195,275.121,-75.042,-178.190,10.207,149.550
C03584=1111.200,274.873,-75.012,-178.193,10.204,149.550
C03585=1111.204,274.625,-74.981,-178.196,10.201,149.550
C03586=1111.208,274.377,-74.952,-178.199,10.198,149.551
C03587=1111.212,274.129,-74.922,-178.201,10.197,149.551
C03588=1111.216,273.881,-74.892,-178.204,10.194,149.551
C03589=1111.221,273.633,-74.862,-178.207,10.191,149.551
C03590=1111.225,273.384,-74.832,-178.210,10.188,149.551
C03591=1111.228,273.136,-74.802,-178.213,10.186,149.551
C03592=1111.233,272.888,-74.771,-178.216,10.183,149.551
C03593=1111.238,272.639,-74.742,-178.219,10.180,149.551
C03594=1111.241,272.392,-74.712,-178.222,10.178,149.552
C03595=1111.246,272.143,-74.682,-178.224,10.176,149.552
C03596=1111.250,271.895,-74.652,-178.227,10.173,149.552
C03597=1111.254,271.647,-74.622,-178.230,10.170,149.552
C03598=1111.259,271.399,-74.593,-178.233,10.167,149.552
C03599=1111.262,271.151,-74.563,-178.236,10.164,149.552
C03600=1111.267,270.903,-74.533,-178.239,10.162,149.552
C03601=1111.271,270.654,-74.503,-178.241,10.160,149.552
C03602=1111.275,270.405,-74.473,-178.244,10.157,149.552
C03603=1111.279,270.158,-74.443,-178.247,10.154,149.552
C03604=1111.283,269.910,-74.414,-178.250,10.151,149.553
C03605=1111.287,269.661,-74.384,-178.253,10.149,149.553
C03606=1111.291,269.449,-74.359,-178.255,10.147,149.553
C03607=1111.294,269.236,-74.333,-178.258,10.145,149.553
C03608=1111.299,269.024,-74.308,-178.260,10.143,149.553
C03609=1111.302,268.811,-74.282,-178.263,10.140,149.553
C03610=1111.306,268.599,-74.257,-178.265,10.138,149.553
C03611=1111.309,268.385,-74.231,-178.267,10.136,149.553
C03612=1111.313,268.173,-74.206,-178.269,10.134,149.553
C03613=1111.316,267.960,-74.180,-178.272,10.132,149.553
C03614=1111.321,267.712,-74.150,-178.275,10.129,149.554
C03615=1111.325,267.464,-74.121,-178.277,10.126,149.554
C03616=1111.329,267.216,-74.092,-178.280,10.123,149.554
C03617=1111.334,266.968,-74.062,-178.283,10.122,149.554
C03618=1111.338,266.720,-74.033,-178.286,10.119,149.554
C03619=1111.342,266.472,-74.004,-178.289,10.116,149.554
C03620=1111.346,266.223,-73.974,-178.292,10.114,149.554
C03621=1111.351,265.975,-73.945,-178.294,10.112,149.554
C03622=1111.355,265.727,-73.915,-178.297,10.109,149.555
C03623=1111.359,265.479,-73.886,-178.300,10.106,149.555
C03624=1111.363,265.230,-73.856,-178.302,10.104,149.555
C03625=1111.367,264.982,-73.827,-178.305,10.101,149.555
C03626=1111.371,264.734,-73.797,-178.308,10.099,149.555
C03627=1111.376,264.485,-73.768,-178.311,10.096,149.555
C03628=1111.380,264.237,-73.738,-178.314,10.093,149.555
C03629=1111.384,263.989,-73.709,-178.318,10.091,149.556
C03630=1111.388,263.741,-73.680,-178.320,10.088,149.556
C03631=1111.392,263.492,-73.650,-178.323,10.085,149.556
C03632=1111.397,263.245,-73.621,-178.326,10.082,149.556
C03633=1111.401,262.997,-73.592,-178.329,10.080,149.556
C03634=1111.405,262.748,-73.562,-178.333,10.077,149.556
C03635=1111.410,262.500,-73.533,-178.335,10.075,149.556
C03636=1111.414,262.251,-73.504,-178.338,10.072,149.556
C03637=1111.418,262.003,-73.474,-178.341,10.070,149.557
C03638=1111.422,261.755,-73.445,-178.344,10.067,149.557
C03639=1111.427,261.506,-73.416,-178.347,10.064,149.557
C03640=1111.431,261.259,-73.387,-178.350,10.061,149.557
C03641=1111.435,261.010,-73.358,-178.353,10.059,149.557
C03642=1111.439,260.762,-73.329,-178.356,10.056,149.557
C03643=1111.444,260.514,-73.299,-178.358,10.053,149.557
C03644=1111.448,260.265,-73.270,-178.361,10.050,149.557
C03645=1111.452,260.016,-73.241,-178.364,10.048,149.557
C03646=1111.456,259.769,-73.213,-178.367,10.044,149.557
C03647=1111.460,259.521,-73.183,-178.370,10.042,149.557
C03648=1111.465,259.272,-73.155,-178.373,10.039,149.558
C03649=1111.469,259.024,-73.125,-178.376,10.036,149.558
C03650=1111.473,258.776,-73.096,-178.379,10.033,149.558
C03651=1111.478,258.528,-73.068,-178.382,10.031,149.558
